(* Logix 5000 project; controller CLASE_1 Emulate 5570 rev 28.11; software revision 28.02; part 13 of 15 *)
(* tags used below, declared in another part *)
   Ref_FaultCodeList : P_DescList[1];   // Tag containing List of Fault Codes (DINT) and their Descriptions (STRING)
   Inp_LastFaultCode : DINT;   // Most recent drive fault code (enumeration)
   Inp_Ready : BOOL;   // 1=Drive is ready to run
   Inp_CommandDir : BOOL;   // 1=Drive is commanded Forward, 0=Drive is commanded Reverse
   Inp_ActualDir : BOOL;   // 1=Drive is running Forward, 0=Drive is running Reverse
   Inp_FwdPermOK : BOOL;   // 1=Permissives OK, drive can start Forward
   Inp_FwdNBPermOK : BOOL;   // 1=Non-Bypassable Permissives OK, drive can start Forward
   Inp_RevPermOK : BOOL;   // 1=Permissives OK, drive can start Reverse
   Inp_RevNBPermOK : BOOL;   // 1=Non-Bypassable Permissives OK, motor can start Reverse
   Inp_IntlkOK : BOOL;   // 1=Interlocks OK, drive can start/run
   Inp_NBIntlkOK : BOOL;   // 1=Non-Bypassable Interlocks OK, drive can start/run
   Inp_IOFault : BOOL;   // Input Communication Status 0=OK, 1=fail
   Inp_Sim : BOOL;   // 1=Simulate working drive; 0=Start/Stop/ Monitor actual drive
   Inp_OvrdCmd : SINT;   // Override Mode Command: 0=None, 1=Stop, 2=Start Fwd 3=Start Rev
   Cfg_HasJog : BOOL;   // 1=Drive Jog Command enabled/visible, 0=Drive Jog Command not allowed
   Cfg_HasRunFdbk : BOOL;   // 1=Drive provides feedback signal on Inp_Running when running
   Cfg_UseRunFdbk : BOOL;   // 1=Drive run feedback should be used for failure checking
   Cfg_HasSpeedFdbk : BOOL;   // 1=Drive provides speed feedback on Inp_SpeedFdbk
   Cfg_UseSpeedFdbk : BOOL;   // 1=Drive speed determines running state, 0=state determined by drive Active input bit
   Cfg_HasOutDatalink : BOOL;   // 1=A signal is connected to Out_Datalink
   Cfg_SetTrack : BOOL;   // 1=PSets track OSets in Oper, OSets track PSets in Prog, 0=no tracking
   Cfg_SetTrackOvrdHand : BOOL;   // 1=Prog/Oper Settings track Override/Hand speed reference
   Cfg_PCmdClear : ALIAS FOR Mode.Cfg_PCmdClear;
   Cfg_ProgDefault : ALIAS FOR Mode.Cfg_ProgDefault;
   Cfg_OperStopPrio : BOOL;   // 1=OCmd_Stop has priority, accepted any time, 0=OCmd_Stop only in Oper, Maint Mode.
   Cfg_OCmdResets : BOOL;   // 1=New Oper drive cmd. resets fault, 0=reset req'd to clear fault
   Cfg_ShedOnFailToStart : BOOL;   // 1=Stop Motor and Alarm on Fail to Start; 0=Alarm only on Fail to Start
   Cfg_ShedOnIOFault : BOOL;   // 1=Stop Motor and Alarm on I/O Fault; 0=Alarm only on I/O Fault
   Cfg_FailToStartAckReqd : ALIAS FOR FailToStart.Cfg_AckReqd;   // 1=Acknowledge required for Fail to Start Alarm
   Cfg_FailToStopAckReqd : ALIAS FOR FailToStop.Cfg_AckReqd;   // 1=Acknowledge required for Fail to Stop Alarm
   Cfg_IntlkTripAckReqd : ALIAS FOR IntlkTrip.Cfg_AckReqd;   // 1=Acknowledge required for Interlock Trip Alarm
   Cfg_DriveFaultAckReqd : ALIAS FOR DriveFault.Cfg_AckReqd;   // 1=Acknowledge required for Drive Fault Alarm
   Cfg_IOFaultAckReqd : ALIAS FOR IOFault.Cfg_AckReqd;   // 1=Acknowledge required for I/O Fault Alarm
   Cfg_FailToStartSeverity : ALIAS FOR FailToStart.Cfg_Severity;   // Fail To Start Alarm Severity: 1..250=Low, 251..500=Medium, 501..750=High, 751..1000=Urgent
   Cfg_FailToStopSeverity : ALIAS FOR FailToStop.Cfg_Severity;   // Fail To Stop Alarm Severity: 1..250=Low, 251..500=Medium, 501..750=High, 751..1000=Urgent
   Cfg_IntlkTripSeverity : ALIAS FOR IntlkTrip.Cfg_Severity;   // Interlock Trip Alarm Severity: 1..250=Low, 251..500=Medium, 501..750=High, 751..1000=Urgent
   Cfg_DriveFaultSeverity : ALIAS FOR DriveFault.Cfg_Severity;   // Drive Fault Alarm Severity: 1..250=Low, 251..500=Medium, 501..750=High, 751..1000=Urgent
   Cfg_IOFaultSeverity : ALIAS FOR IOFault.Cfg_Severity;   // I/O Fault Alarm Severity: 1..250=Low, 251..500=Medium, 501..750=High, 751..1000=Urgent
   Cfg_MinSpdRef : REAL;   // Minimum Speed Reference in EU (for limiting)
   Cfg_MaxSpdRef : REAL;   // Maximum Speed Reference in EU (for limiting)
   Cfg_SpeedRefRawMin : REAL;   // Speed Reference Minimum in Drive (raw) Units (for scaling)
   Cfg_SpeedRefRawMax : REAL;   // Speed Reference Maximum in Drive (raw) Units (for scaling)
   Cfg_SpeedRefEUMin : REAL;   // Speed Reference Minimum in Engineering Units (for scaling)
   Cfg_SpeedRefEUMax : REAL;   // Speed Reference Maximum in Engineering Units (for scaling)
   Cfg_SpeedFdbkRawMax : REAL;   // Speed Feedback Maximum in Drive (raw) Units (for scaling)
   Cfg_SpeedFdbkEUMax : REAL;   // Speed Feedback Maximum in Engineering Units (for scaling)
   Cfg_InpDatalinkRawMax : REAL;   // Input Datalink Maximum in Drive (raw) Units (for scaling)
   Cfg_InpDatalinkEUMax : REAL;   // Input Datalink Maximum in Engineering Units (for scaling)
   Cfg_OutDatalinkMax : REAL;   // Maximum Output Datalink in EU (for limiting)
   Cfg_OutDatalinkRawMin : REAL;   // Output Datalink Minimum in Drive (raw) Units (for scaling)
   Cfg_OutDatalinkRawMax : REAL;   // Output Datalink Maximum in Drive (raw) Units (for scaling)
   Cfg_OutDatalinkEUMin : REAL;   // Output Datalink Minimum in Engineering Units (for scaling)
   Cfg_OutDatalinkEUMax : REAL;   // Output Datalink Maximum in Engineering Units (for scaling)
   Cfg_SimRampT : DINT;   // Time to ramp speed fdbk when in Simulation (sec)
   Cfg_FailToStartT : DINT;   // Time after Start to get Run Feedback before Fault (sec)
   Cfg_FailToStopT : DINT;   // Time after Stop to drop Run Feedback before Fault (sec)
   Cfg_ResetPulseT : DINT;   // Time to pulse Out_Reset to clear drive fault
   Cfg_OperKeep : SINT;   // Oper keeps control in Prog Mode: .0=Reference, .1=Start/Stop, .2=Fwd/Rev, .3=OutDatalink
   Cfg_ProgKeep : SINT;   // Prog keeps control in Oper Mode: .0=Reference, .1=Start/Stop, .2=Fwd/Rev, .3=OutDatalink
   PSet_SpeedRef : REAL;   // Program Setting of Speed Reference (EU)
   PSet_OutDatalink : REAL;   // Program Setting of Output Datalink (EU)
   PSet_Owner : DINT;   // Program Owner Request ID (non-zero) or Release (zero)
   OSet_SpeedRef : REAL;   // Operator Setting of Speed Reference (EU)
   OSet_OutDatalink : REAL;   // Operator Setting of Output Datalink (EU)
   PCmd_Start : BOOL;   // Program Command to Start Drive
   PCmd_Stop : BOOL;   // Program Command to Stop Drive
   PCmd_Fwd : BOOL;   // Program Command to set direction to Fowrard
   PCmd_Rev : BOOL;   // Program Command to set direction to Reverse
   PCmd_Reset : BOOL;   // Program Command to Reset drive fault and all Alarms requiring Reset
   OCmd_Start : BOOL;   // Operator Command to Start Drive
   OCmd_Stop : BOOL;   // Operator Command to Stop Drive
   OCmd_Jog : BOOL;   // Operator Command to Jog Drive (not cleared by P_VSD!)
   OCmd_Fwd : BOOL;   // Operator Command to set direction to Forward
   OCmd_Rev : BOOL;   // Operator Command to set direction to Reverse
   OCmd_Bypass : BOOL;   // Operator Command to Bypass all Bypassable Interlocks and Permissives
   OCmd_Check : BOOL;   // Operator Command to Check (not bypass) all Interlocks and Permissives
   MCmd_Disable : BOOL;   // Maintenance Command to Disable Drive
   MCmd_Enable : BOOL;   // Maintenance Command to Enable (allow to run) Drive
   OCmd_Reset : BOOL;   // Operator Command to Reset all Alarms requiring Reset
   OCmd_ResetAckAll : BOOL;   // Operator Command to Reset all Alarms and latched Shed conditions
   Out_SpeedRef : REAL;   // Drive Speed Reference in Drive Units (typ. 0-32767 = 0 to max freq.)
   Out_Datalink : REAL;   // Auxiliary Signal (datalink) Output in Drive (raw) Units
   Out_Run : BOOL;   // 1=Start/Run Drive, 0=Stop Drive (for held starter type)
   Out_Stop : BOOL;   // 1=Stop Drive, 0=drive left in current state
   Out_Start : BOOL;   // 1=Start Drive, 0=drive left in current state
   Out_Jog : BOOL;   // 1=Jog drive at Jog Speed, -->0=stop jogging
   Out_ClearFault : BOOL;   // 1=Attempt to clear Drive Fault
   Out_Fwd : BOOL;   // 1=Set drive direction to Forward
   Out_Rev : BOOL;   // 1=Set drive direction to Reverse
   Val_SpeedRef : REAL;   // Speed Reference (target) to drive
   Val_OutDatalink : REAL;   // Output Datalink value to drive
   Val_SpeedRefEUMax : REAL;   // Maximum of Speed Reference = MAX (Cfg_SpeedFdbkEUMin, Cfg_SpeedFdbkEUMax)
   Val_SpeedFdbkEUMax : REAL;   // Maximum of Speed Feedback = MAX (Cfg_SpeedFdbkEUMin, Cfg_SpeedFdbkEUMax)
   Val_LastFaultCode : DINT;   // Most recent drive fault code (enumeration)
   SrcQ_IO : SINT;   // Source and Quality of primary I/O (enumeration)
   SrcQ : SINT;   // Source and Quality of primary Val/Sts (enumeration)
   Val_Cmd : SINT;   // Device Command 0=None, 1=Stop, 2=StartFwd 3=StartRev 4=JogFwd 5=JogRev
   Val_Fdbk : SINT;   // Device Feedback 0=Stopped, 1=Running Fwd 2=Running Rev 3=Accelerating 4=Decelerating
   Val_Sts : SINT;   // Device Confirmed Sts 0? 1=Stop 2=RunF 3=RunR 4=JogF 5=JogR 6=Stopping 7=Starting F 8=Starting R, 33=Disabled
   Val_Fault : SINT;   // Device Fault Status 0=None, 16=Fail to Start, 17 = Fail to Stop, 18=Drive Fault, 32=I/O Fault, 34=Config Error
   Val_Mode : ALIAS FOR Mode.Val;
   Val_Owner : DINT;   // Current Object Owner ID (0=not owned)
   Val_Notify : SINT;   // Current Alarm Level and Acknowledgement (enumeration)
   Sts_Stopped : BOOL;   // 1=Drive requested to stop and is confirmed stopped
   Sts_Starting : BOOL;   // 1=Drive requested to run and awaiting run feedback
   Sts_Running : BOOL;   // 1=Drive requested to run and is confirmed running
   Sts_Stopping : BOOL;   // 1=Drive requested to stop and awaiting stopped feedback
   Sts_Jogging : BOOL;   // 1=Drive requested to Jog
   Sts_CommandDir : BOOL;   // 1=Drive commanded to Forward, 0=Reverse
   Sts_ActualDir : BOOL;   // 1=Drive Actual direction is Forward, 0=Reverse
   Sts_SpeedLimited : BOOL;   // 1=Speed Reference Setting exceeds configured Max/Min limit
   Sts_Disabled : BOOL;   // 1=Drive is Disabled
   Sts_NotRdy : BOOL;   // 1=Device Not Ready, see detail bits for reason
   Nrdy_OperPrio : BOOL;   // 1=Device Not Ready: Operator State 0 Priority Command Requires Reset
   Nrdy_Fail : BOOL;   // 1=Device Not Ready: Device Failure (Shed Requires Reset)
   Nrdy_IOFault : BOOL;   // 1=Device Not Ready: I/O Fault (Shed Requires Reset)
   Nrdy_Trip : BOOL;   // 1=Device not Ready: Deivce Tripped (Drive Fault)
   Sts_AlmInh : BOOL;   // 1=An Alarm is Shelved, Disabled or Suppressed, display icon
   Sts_Err : BOOL;   // 1=Error in Config: see detail bits for reason
   Err_FdbkRaw : BOOL;   // 1=Erron in Config: Speed Fdbk Raw Min = Max
   Err_FdbkEU : BOOL;   // 1=Error in Config: Speed Fdbk EU Min = Max
   Err_RefEU : BOOL;   // 1=Error in Config: Speed Ref EU Min = Max
   Err_OutDLEU : BOOL;   // 1=Error in Config: Output Datalink EU Min = Max
   Sts_Hand : ALIAS FOR Mode.Sts_Hand;
   Sts_Maint : ALIAS FOR Mode.Sts_Maint;
   Sts_Ovrd : ALIAS FOR Mode.Sts_Ovrd;
   Sts_Prog : ALIAS FOR Mode.Sts_Prog;
   Sts_Oper : ALIAS FOR Mode.Sts_Oper;
   Ack_FailToStart : ALIAS FOR FailToStart.Ack;   // 1=Fail to Start Alarm has been acknowledged
   Sts_FailToStop : ALIAS FOR FailToStop.Inp;   // 1=Drive Failed to Stop
   Ack_FailToStop : ALIAS FOR FailToStop.Ack;   // 1=Fail to Stop Alarm has been acknowledged
   Ack_IntlkTrip : ALIAS FOR IntlkTrip.Ack;   // 1=Interlock Trip Alarm has been acknowledged
   Sts_DriveFault : ALIAS FOR DriveFault.Inp;   // 1=Drive Fault (see drive display or manual)
   Ack_DriveFault : ALIAS FOR DriveFault.Ack;   // 1=Drive Fault Alarm has been acknowledged
   Sts_IOFault : ALIAS FOR IOFault.Inp;   // I/O Comm Fault Status (0=OK, 1=Bad)
   Ack_IOFault : ALIAS FOR IOFault.Ack;   // 1=I/O Fault Alarm has been acknowledged
   Rdy_Start : BOOL;   // 1=Ready to receive OCmd_Start (enables HMI button)
   Rdy_Stop : BOOL;   // 1=Ready to receive OCmd_Stop (enables HMI button)
   Rdy_Jog : BOOL;   // 1=Ready to receive OCmd_Jog (enables HMI button)
   Rdy_Bypass : BOOL;   // 1=Ready to receive OCmd_Bypass (enables HMI button)
   Rdy_Reset : BOOL;   // 1=Ready to receive OCmd_Reset (enables HMI button)
   Rdy_ResetAckAll : BOOL;   // 1=At least one Alarm or latched Shed condition requires Reset or Ack
   Rdy_SpeedRef : BOOL;   // 1=Ready to receive OSet_SpeedRef (enables data entry field)
   Rdy_OSet : BOOL;   // 1=Ready to receive OSets (other than CV) (enables data entry fields)
   P_VSD : BOOL;   // Unique Parameter Name for auto - discovery
   Mode : P_Mode;   // Drive Mode Selection
   IOFault : P_Alarm;   // I/O Fault Alarm
   IntlkTrip : P_Alarm;   // Interlock Trip Alarm
   FailToStop : P_Alarm;   // Drive Failed to Stop Alarm
   FailToStart : P_Alarm;   // Drive Failed to Start Alarm
   Wrk_Run : BOOL;   // 1=Drive should be "running", 0=should be "stopped"
   Wrk_RunFdbk : BOOL;   // Run Feedback based on mode, simulation, etc. 1=running
   Wrk_Notify : DINT;   // Buffer for building Val_Notify
   DriveFault : P_Alarm;   // Drive Faulted Alarm
   Wrk_SpeedRef : REAL;   // Working copy of Speed Reference (for limiting)
   Wrk_Rev : BOOL;   // Working (internal) Direction 1=Reverse 0=Forward (default)
   Wrk_Jog : BOOL;   // 1=Jog Drive, 0=Drive not jogging
   Wrk_OutDatalink : REAL;   // Selected Output Datalink setting
   Wrk_Cmd : SINT;   // Buffer for building Val_Cmd
   Wrk_Sts : SINT;   // Buffer for building Val_Sts
   Wrk_Fault : SINT;   // Buffer for building Val_Fault
   Wrk_Retrigger : BOOL;   // Maint Start issued while running or Stop while stopped
   Wrk_FaultDescFSC : CONTROL;   // FSC control for Fault Code List search
   Val_FaultDesc : STRING_40;   // Description of Drive Fault (given LastFaultCode)
   Wrk_SrcQ : SINT;   // Register for building Source / Quality enumeration
   Wrk_NotRdy : BOOL;   // Device Not Ready conditions excluding shed latches
(* P_VSD, continued *)

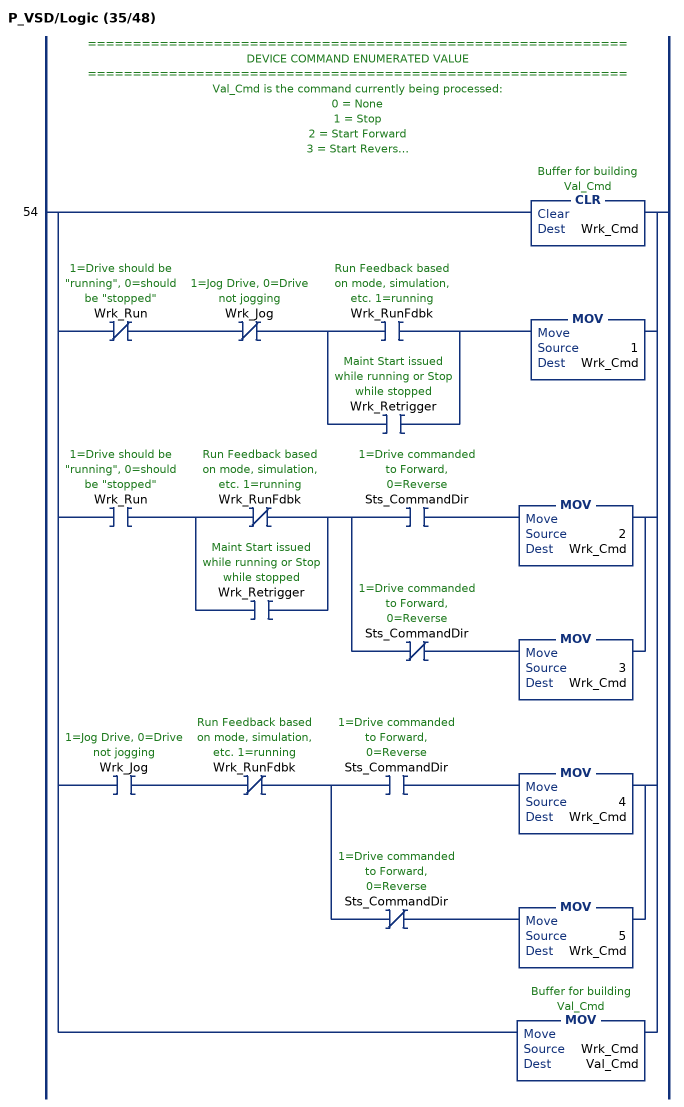
   [picture p271: P_VSD/Logic rungs 54-54]
   // ============================================================
   // DEVICE COMMAND ENUMERATED VALUE
   // ============================================================
   // Val_Cmd is the command currently being processed:
   // 0 = None
   // 1 = Stop
   // 2 = Start Forward
   // 3 = Start Reverse
   // 4 = Jog Forward
   // 5 = Jog Reverse
   54: [CLR(Wrk_Cmd) ,XIO(Wrk_Run) XIO(Wrk_Jog) [XIC(Wrk_RunFdbk) ,XIC(Wrk_Retrigger) ] MOV(1,Wrk_Cmd) ,XIC(Wrk_Run) [XIO(Wrk_RunFdbk) ,XIC(Wrk_Retrigger) ] [XIC(Sts_CommandDir) MOV(2,Wrk_Cmd) ,XIO(Sts_CommandDir) MOV(3,Wrk_Cmd) ] ,XIC(Wrk_Jog) XIO(Wrk_RunFdbk) [XIC(Sts_CommandDir) MOV(4,Wrk_Cmd) ,XIO(Sts_CommandDir) MOV(5,Wrk_Cmd) ] ,MOV(Wrk_Cmd,Val_Cmd) ];
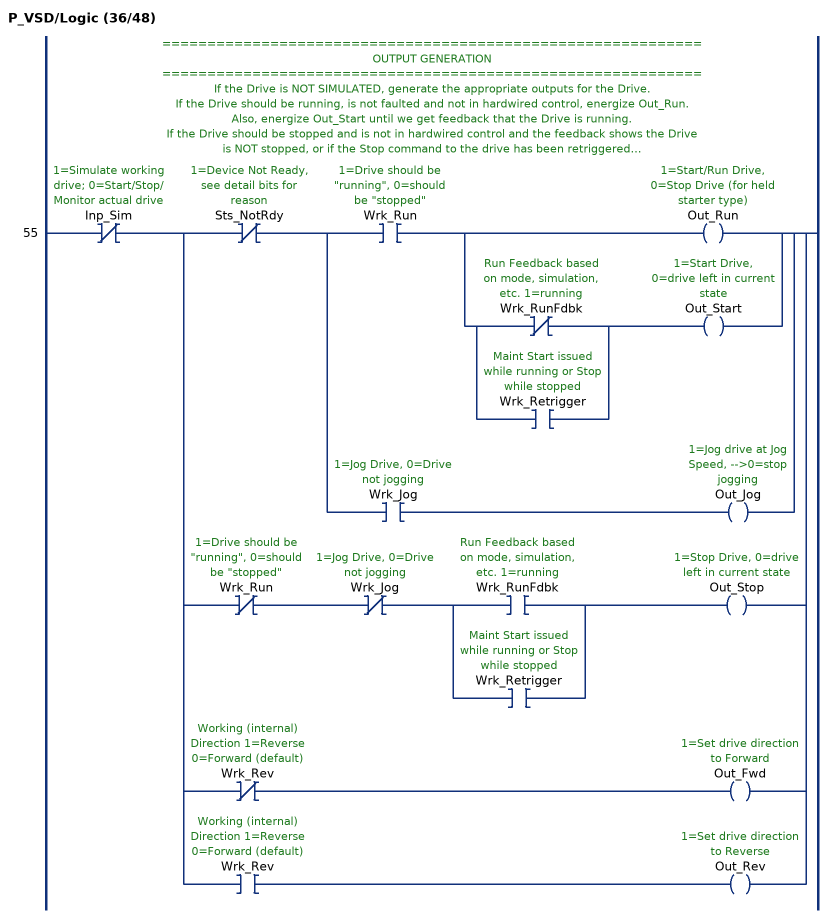
   // ============================================================
   // OUTPUT GENERATION
   // ============================================================
   // If the Drive is NOT SIMULATED, generate the appropriate outputs for the Drive.
   // If the Drive should be running, is not faulted and not in hardwired control, energize Out_Run.
   // Also, energize Out_Start until we get feedback that the Drive is running.
   // If the Drive should be stopped and is not in hardwired control and the feedback shows the Drive
   // is NOT stopped, or if the Stop command to the drive has been retriggered,
   // energize the Out_Stop output to stop the Drive.
   // Finally, if the drive is not simulated, energize the appropriate direction output.
   // #####  V3.5-02  2016-03-22:  Modified to eliminate oscillating Out_Stop on Drive Not Ready.  #####
   55: XIO(Inp_Sim)[XIO(Sts_NotRdy) [XIC(Wrk_Run) [OTE(Out_Run) ,[XIO(Wrk_RunFdbk) ,XIC(Wrk_Retrigger) ] OTE(Out_Start) ] ,XIC(Wrk_Jog) OTE(Out_Jog) ] ,XIO(Wrk_Run) XIO(Wrk_Jog) [XIC(Wrk_RunFdbk) ,XIC(Wrk_Retrigger) ] OTE(Out_Stop) ,XIO(Wrk_Rev) OTE(Out_Fwd) ,XIC(Wrk_Rev) OTE(Out_Rev) ];
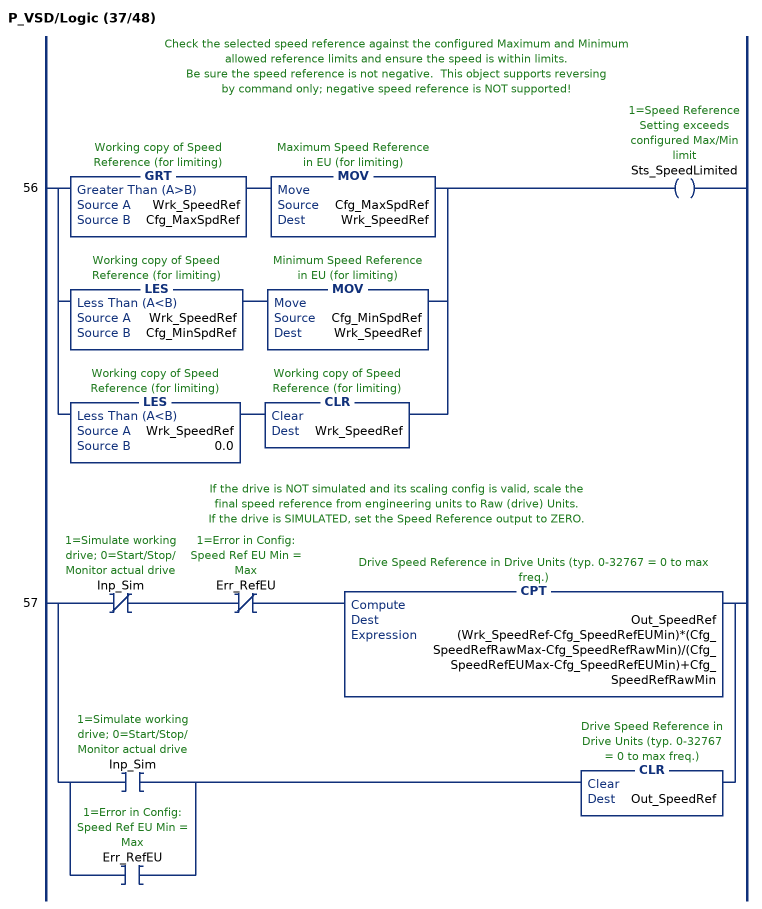
   // Check the selected speed reference against the configured Maximum and Minimum
   // allowed reference limits and ensure the speed is within limits.
   // Be sure the speed reference is not negative.  This object supports reversing
   // by command only; negative speed reference is NOT supported!
   56: [GRT(Wrk_SpeedRef,Cfg_MaxSpdRef) MOV(Cfg_MaxSpdRef,Wrk_SpeedRef) ,LES(Wrk_SpeedRef,Cfg_MinSpdRef) MOV(Cfg_MinSpdRef,Wrk_SpeedRef) ,LES(Wrk_SpeedRef,0.0) CLR(Wrk_SpeedRef) ]OTE(Sts_SpeedLimited);
   // If the drive is NOT simulated and its scaling config is valid, scale the
   // final speed reference from engineering units to Raw (drive) Units.
   // If the drive is SIMULATED, set the Speed Reference output to ZERO.
   57: [XIO(Inp_Sim) XIO(Err_RefEU) CPT(Out_SpeedRef,(Wrk_SpeedRef-Cfg_SpeedRefEUMin)*(Cfg_SpeedRefRawMax-Cfg_SpeedRefRawMin)/(Cfg_SpeedRefEUMax-Cfg_SpeedRefEUMin)+Cfg_SpeedRefRawMin) ,[XIC(Inp_Sim) ,XIC(Err_RefEU) ] CLR(Out_SpeedRef) ];
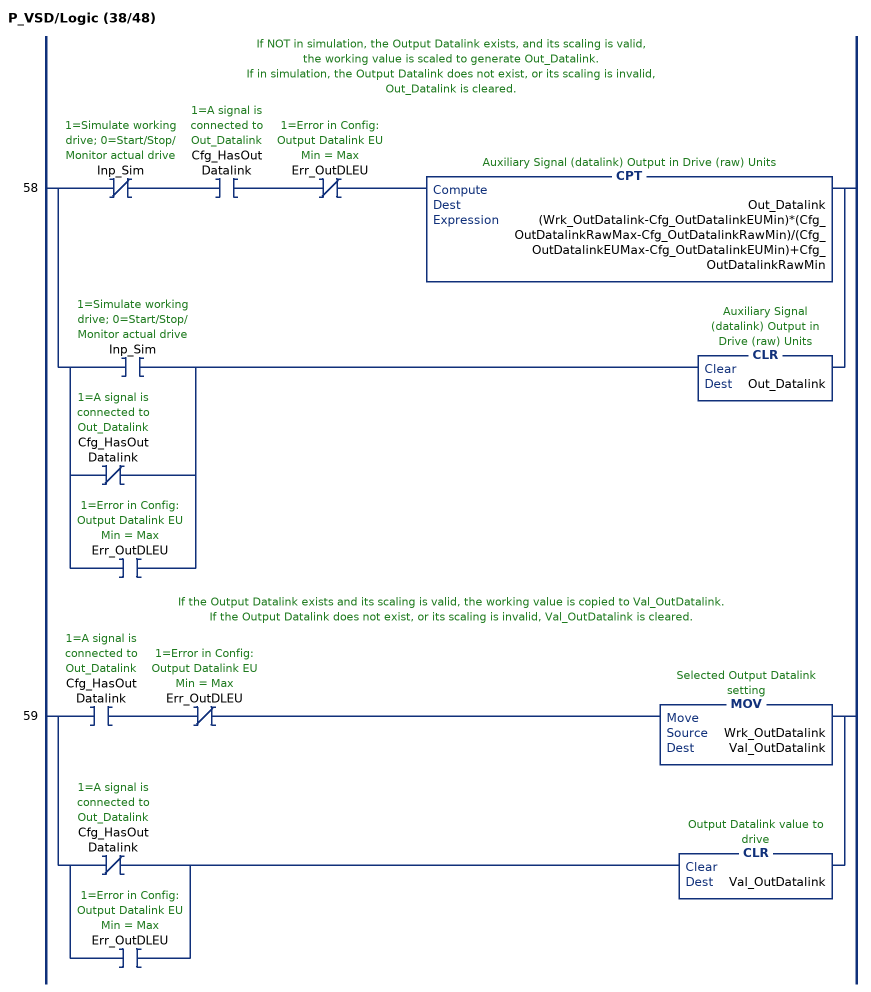
   // If NOT in simulation, the Output Datalink exists, and its scaling is valid,
   // the working value is scaled to generate Out_Datalink.
   // If in simulation, the Output Datalink does not exist, or its scaling is invalid,
   // Out_Datalink is cleared.
   58: [XIO(Inp_Sim) XIC(Cfg_HasOutDatalink) XIO(Err_OutDLEU) CPT(Out_Datalink,(Wrk_OutDatalink-Cfg_OutDatalinkEUMin)*(Cfg_OutDatalinkRawMax-Cfg_OutDatalinkRawMin)/(Cfg_OutDatalinkEUMax-Cfg_OutDatalinkEUMin)+Cfg_OutDatalinkRawMin) ,[XIC(Inp_Sim) ,XIO(Cfg_HasOutDatalink) ,XIC(Err_OutDLEU) ] CLR(Out_Datalink) ];
   // If the Output Datalink exists and its scaling is valid, the working value is copied to Val_OutDatalink.
   // If the Output Datalink does not exist, or its scaling is invalid, Val_OutDatalink is cleared.
   59: [XIC(Cfg_HasOutDatalink) XIO(Err_OutDLEU) MOV(Wrk_OutDatalink,Val_OutDatalink) ,[XIO(Cfg_HasOutDatalink) ,XIC(Err_OutDLEU) ] CLR(Val_OutDatalink) ];
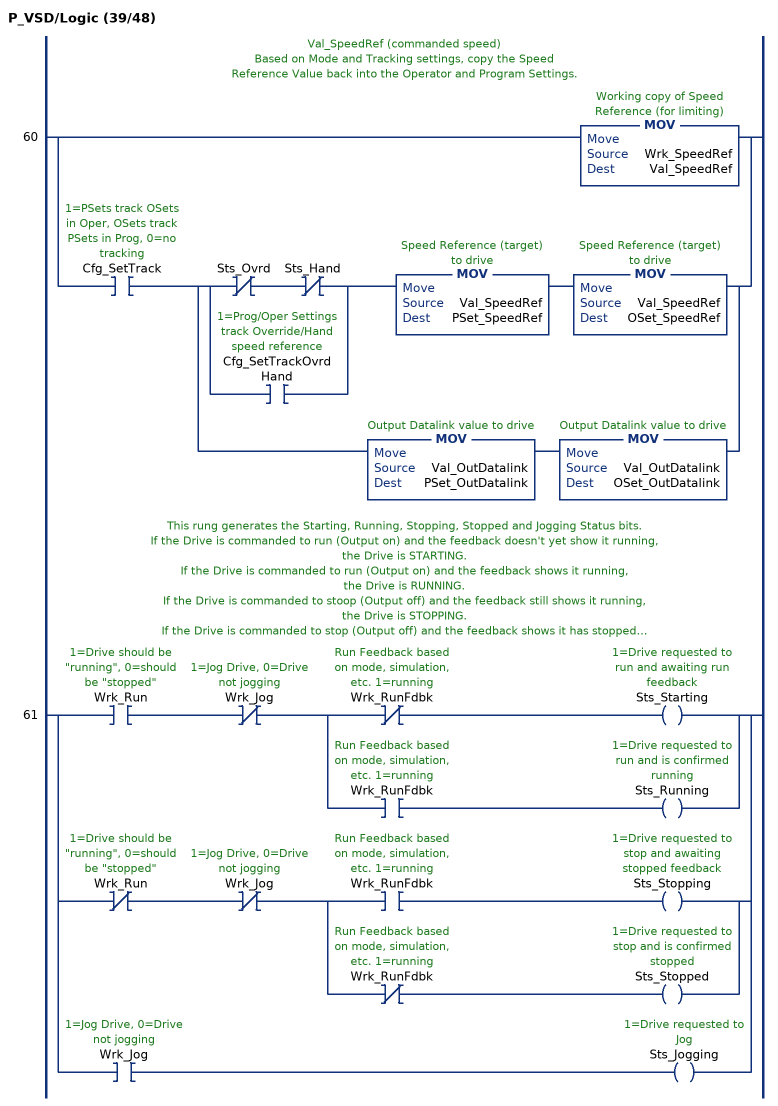
   // Val_SpeedRef (commanded speed)
   // Based on Mode and Tracking settings, copy the Speed
   // Reference Value back into the Operator and Program Settings.
   60: [MOV(Wrk_SpeedRef,Val_SpeedRef) ,XIC(Cfg_SetTrack) [[XIO(Sts_Ovrd) XIO(Sts_Hand) ,XIC(Cfg_SetTrackOvrdHand) ] MOV(Val_SpeedRef,PSet_SpeedRef) MOV(Val_SpeedRef,OSet_SpeedRef) ,MOV(Val_OutDatalink,PSet_OutDatalink) MOV(Val_OutDatalink,OSet_OutDatalink) ] ];
   // This rung generates the Starting, Running, Stopping, Stopped and Jogging Status bits.
   // If the Drive is commanded to run (Output on) and the feedback doesn't yet show it running,
   // the Drive is STARTING.
   // If the Drive is commanded to run (Output on) and the feedback shows it running,
   // the Drive is RUNNING.
   // If the Drive is commanded to stoop (Output off) and the feedback still shows it running,
   // the Drive is STOPPING.
   // If the Drive is commanded to stop (Output off) and the feedback shows it has stopped,
   // the Drive is STOPPED.
   // #####  V3.0-00  2013-06-30:  Removed check of Cfg_UseRunFdbk --  #####
   // #####  now uses run feedback  based on speed fdbk  #####
   61: [XIC(Wrk_Run) XIO(Wrk_Jog) [XIO(Wrk_RunFdbk) OTE(Sts_Starting) ,XIC(Wrk_RunFdbk) OTE(Sts_Running) ] ,XIO(Wrk_Run) XIO(Wrk_Jog) [XIC(Wrk_RunFdbk) OTE(Sts_Stopping) ,XIO(Wrk_RunFdbk) OTE(Sts_Stopped) ] ,XIC(Wrk_Jog) OTE(Sts_Jogging) ];
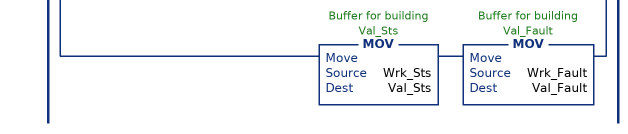
   // Val_Sts is the current device status, as determined by this AOI,
   // based on its knowledge of commands executed and feedback.
   // (This is the status that should be monitored by, for example, FT Historian.)
   // 0 = Powerup / Unknown (Hand Mode with no feedback, for example)
   // 1 = Stopped
   // 2 = Running Forward
   // 3 = Running Reverse
   // 4 = Jogging Forward
   // 5 = Jogging Reverse
   // 6 = Stopping
   // 7 = Starting Forward
   // 8 = Starting Reverse
   // 33 = Device Disabled
   // Val_Fault is the current device fault status, as determined by this AOI,
   // based on its knowledge of commands executed and feedback.
   // (This is the fault status that should be monitored by, for example, FT Historian.)
   // 0 = None
   // 16 = Fail to Start
   // 17 = Fail to Stop
   // 18 = Drive Fault
   // 32 = I/O Fault (from Input)
   // 34 = Configuration Error
   // #####  V3.1-00  2014-06-30: Added Not Ready reason bits (Nrdy_xxx)  #####
   62: [CLR(Wrk_Sts) CLR(Wrk_Fault) ,XIC(Sts_Stopped) MOV(1,Wrk_Sts) ,XIC(Sts_Running) [XIC(Sts_ActualDir) MOV(2,Wrk_Sts) ,XIO(Sts_ActualDir) MOV(3,Wrk_Sts) ] ,XIC(Sts_Jogging) [XIC(Sts_ActualDir) MOV(4,Wrk_Sts) ,XIO(Sts_ActualDir) MOV(5,Wrk_Sts) ] ,XIC(Sts_Stopping) MOV(6,Wrk_Sts) ,XIC(Sts_Starting) [XIC(Sts_CommandDir) MOV(7,Wrk_Sts) ,XIO(Sts_CommandDir) MOV(8,Wrk_Sts) ] ,XIC(Nrdy_Fail) MOV(16,Wrk_Fault) ,XIC(Sts_FailToStop) MOV(17,Wrk_Fault) ,XIC(Sts_DriveFault) MOV(18,Wrk_Fault) ,XIC(Nrdy_IOFault) MOV(32,Wrk_Fault) ,XIC(Sts_Disabled) MOV(33,Wrk_Sts) ,XIC(Sts_Err) MOV(34,Wrk_Fault) ,MOV(Wrk_Sts,Val_Sts) MOV(Wrk_Fault,Val_Fault) ];
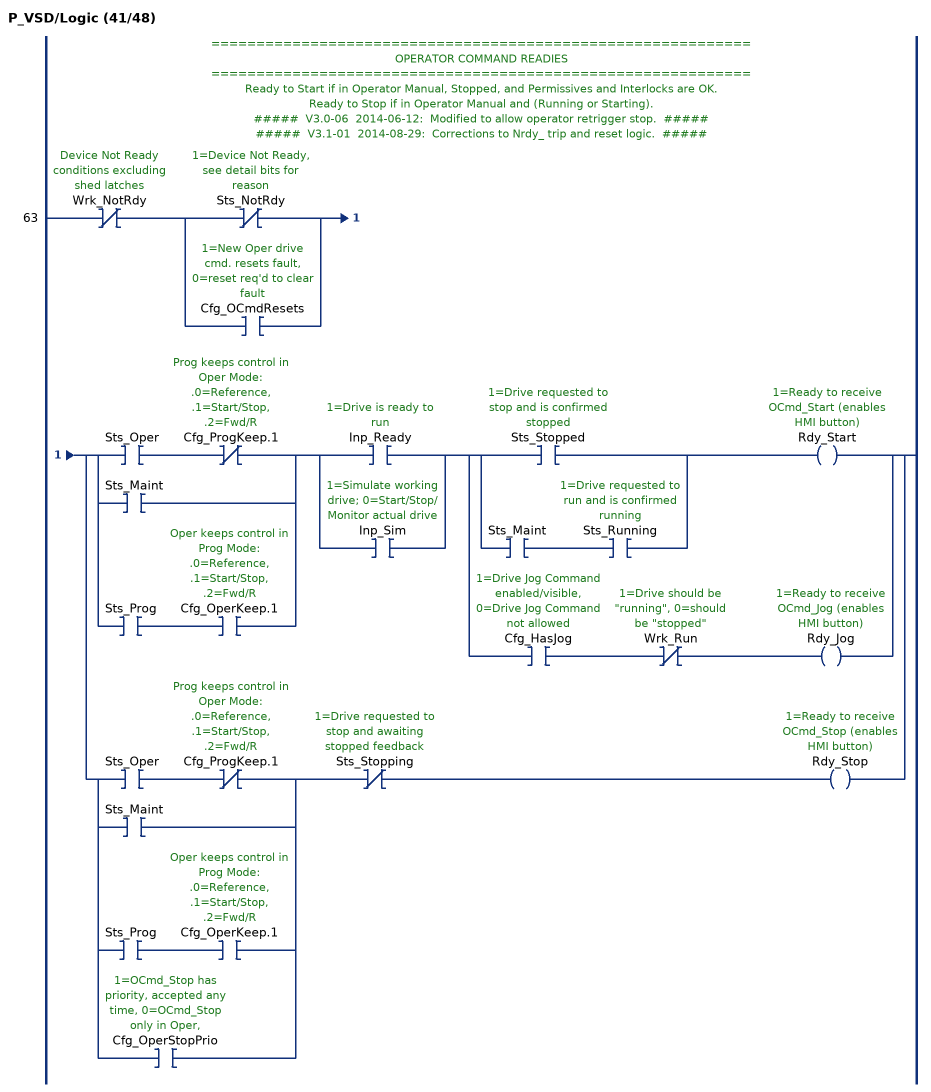
   // ============================================================
   // OPERATOR COMMAND READIES
   // ============================================================
   // Ready to Start if in Operator Manual, Stopped, and Permissives and Interlocks are OK.
   // Ready to Stop if in Operator Manual and (Running or Starting).
   // #####  V3.0-06  2014-06-12:  Modified to allow operator retrigger stop.  #####
   // #####  V3.1-01  2014-08-29:  Corrections to Nrdy_ trip and reset logic.  #####
   63: XIO(Wrk_NotRdy)[XIO(Sts_NotRdy) ,XIC(Cfg_OCmdResets) ][[XIC(Sts_Oper) XIO(Cfg_ProgKeep.1) ,XIC(Sts_Maint) ,XIC(Sts_Prog) XIC(Cfg_OperKeep.1) ] [XIC(Inp_Ready) ,XIC(Inp_Sim) ] [[XIC(Sts_Stopped) ,XIC(Sts_Maint) XIC(Sts_Running) ] OTE(Rdy_Start) ,XIC(Cfg_HasJog) XIO(Wrk_Run) OTE(Rdy_Jog) ] ,[XIC(Sts_Oper) XIO(Cfg_ProgKeep.1) ,XIC(Sts_Maint) ,XIC(Sts_Prog) XIC(Cfg_OperKeep.1) ,XIC(Cfg_OperStopPrio) ] XIO(Sts_Stopping) OTE(Rdy_Stop) ];
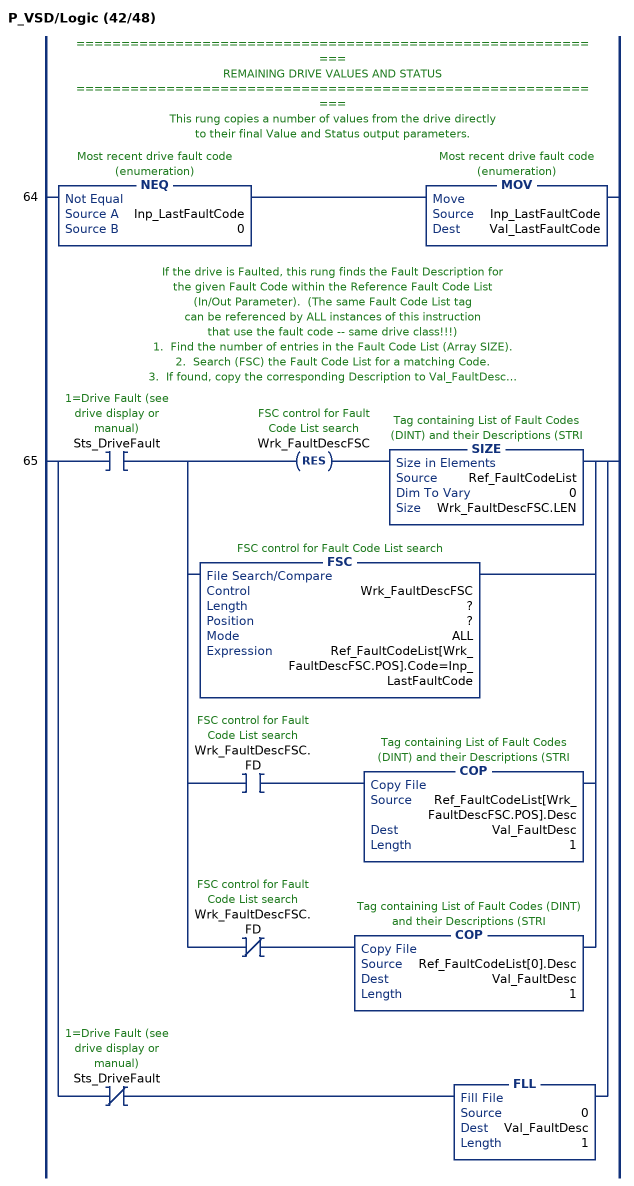
   // ============================================================
   // REMAINING DRIVE VALUES AND STATUS
   // ============================================================
   // This rung copies a number of values from the drive directly
   // to their final Value and Status output parameters.
   64: NEQ(Inp_LastFaultCode,0)MOV(Inp_LastFaultCode,Val_LastFaultCode);
   // If the drive is Faulted, this rung finds the Fault Description for
   // the given Fault Code within the Reference Fault Code List
   // (In/Out Parameter).  (The same Fault Code List tag
   // can be referenced by ALL instances of this instruction
   // that use the fault code -- same drive class!!!)
   // 1.  Find the number of entries in the Fault Code List (Array SIZE).
   // 2.  Search (FSC) the Fault Code List for a matching Code.
   // 3.  If found, copy the corresponding Description to Val_FaultDesc.
   // 4.  If NOT found, copy list entry zero ("No Help Available for this code").
   // And if the drive is not faulted, clear the Val_FaultDesc string.
   // #####  V3.0-00  2013-06-30:  Added rung  #####
   65: [XIC(Sts_DriveFault) [RES(Wrk_FaultDescFSC) SIZE(Ref_FaultCodeList,0,Wrk_FaultDescFSC.LEN) ,FSC(Wrk_FaultDescFSC,?,?,ALL,Ref_FaultCodeList[Wrk_FaultDescFSC.POS].Code=Inp_LastFaultCode) ,XIC(Wrk_FaultDescFSC.FD) COP(Ref_FaultCodeList[Wrk_FaultDescFSC.POS].Desc,Val_FaultDesc,1) ,XIO(Wrk_FaultDescFSC.FD) COP(Ref_FaultCodeList[0].Desc,Val_FaultDesc,1) ] ,XIO(Sts_DriveFault) FLL(0,Val_FaultDesc,1) ];
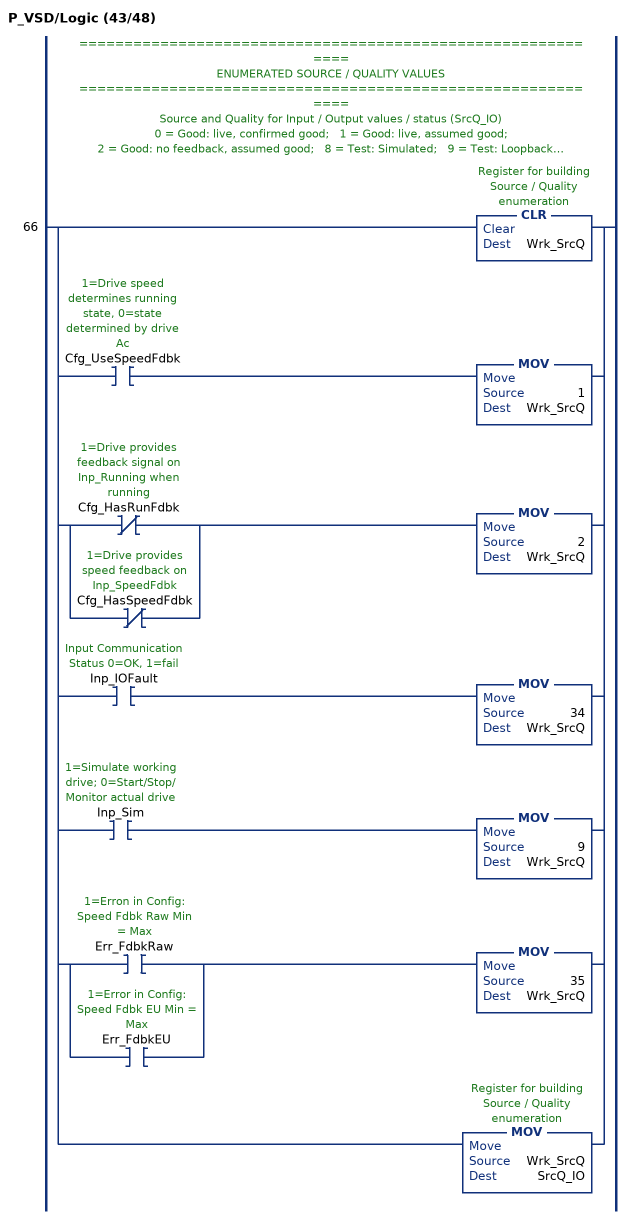
   // ============================================================
   // ENUMERATED SOURCE / QUALITY VALUES
   // ============================================================
   // Source and Quality for Input / Output values / status (SrcQ_IO)
   // 0 = Good: live, confirmed good;   1 = Good: live, assumed good;
   // 2 = Good: no feedback, assumed good;   8 = Test: Simulated;   9 = Test: Loopback;
   // 10 = Test: Manually Entered;   16 = Uncertain: Live, off-spec;
   // 17 = Uncertain, Substituted at Device / Bus;   18 = Uncertain, Substituted at AOI;
   // 19 = Uncertain, using last known good;    20 = Uncertain, using replacement value;
   // 32 = Bad, Signal Failure;   33 = Bad, Channel Fault;
   // 34 = Bad, Module / Comms Fault;   35 = Bad, Invalid Configuration
   // #####  V3.1-00  2014-06-30:  Added rung for Source/Quality enumerations.  #####
   // #####  V3.1-04 Patch01  2015-09-25:  Modified for correct meaning / handling of  #####
   // #####  Cfg_UseSpeedFdbk = 1 (state determined by speed), Cfg_HasRunFdbk = 0  #####
   // #####  (state assumed), and Cfg_HasSpeedFdbk = 0 (speed assumed, no feedback).  #####
   66: [CLR(Wrk_SrcQ) ,XIC(Cfg_UseSpeedFdbk) MOV(1,Wrk_SrcQ) ,[XIO(Cfg_HasRunFdbk) ,XIO(Cfg_HasSpeedFdbk) ] MOV(2,Wrk_SrcQ) ,XIC(Inp_IOFault) MOV(34,Wrk_SrcQ) ,XIC(Inp_Sim) MOV(9,Wrk_SrcQ) ,[XIC(Err_FdbkRaw) ,XIC(Err_FdbkEU) ] MOV(35,Wrk_SrcQ) ,MOV(Wrk_SrcQ,SrcQ_IO) ];
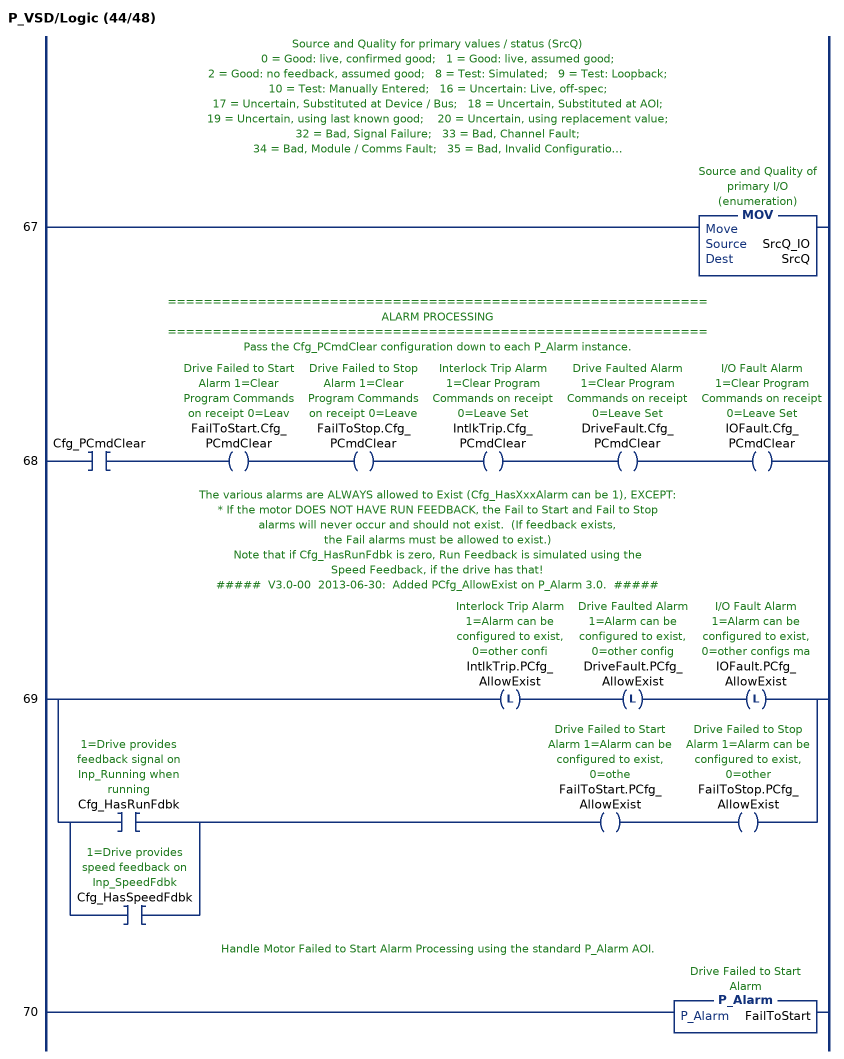
   // Source and Quality for primary values / status (SrcQ)
   // 0 = Good: live, confirmed good;   1 = Good: live, assumed good;
   // 2 = Good: no feedback, assumed good;   8 = Test: Simulated;   9 = Test: Loopback;
   // 10 = Test: Manually Entered;   16 = Uncertain: Live, off-spec;
   // 17 = Uncertain, Substituted at Device / Bus;   18 = Uncertain, Substituted at AOI;
   // 19 = Uncertain, using last known good;    20 = Uncertain, using replacement value;
   // 32 = Bad, Signal Failure;   33 = Bad, Channel Fault;
   // 34 = Bad, Module / Comms Fault;   35 = Bad, Invalid Configuration
   // If the drive is using run feedback (for state) and has speed feedback, all is live and good.
   // If the drive is using speed feedback to determine run state, state is assumed good.
   // If the drive does not have speed feedback, speed is no-feedback assumed good.
   // #####  V3.1-00  2014-06-30:  Added rung for Source/Quality enumerations.  #####
   // #####  V3.1-04 Patch01  2015-09-25:  Modified: instruction does not have substitution of speed feedback.  #####
   67: MOV(SrcQ_IO,SrcQ);
   // ============================================================
   // ALARM PROCESSING
   // ============================================================
   // Pass the Cfg_PCmdClear configuration down to each P_Alarm instance.
   68: XIC(Cfg_PCmdClear)OTE(FailToStart.Cfg_PCmdClear)OTE(FailToStop.Cfg_PCmdClear)OTE(IntlkTrip.Cfg_PCmdClear)OTE(DriveFault.Cfg_PCmdClear)OTE(IOFault.Cfg_PCmdClear);
   // The various alarms are ALWAYS allowed to Exist (Cfg_HasXxxAlarm can be 1), EXCEPT:
   // * If the motor DOES NOT HAVE RUN FEEDBACK, the Fail to Start and Fail to Stop
   // alarms will never occur and should not exist.  (If feedback exists,
   // the Fail alarms must be allowed to exist.)
   // Note that if Cfg_HasRunFdbk is zero, Run Feedback is simulated using the
   // Speed Feedback, if the drive has that!
   // #####  V3.0-00  2013-06-30:  Added PCfg_AllowExist on P_Alarm 3.0.  #####
   69: [OTL(IntlkTrip.PCfg_AllowExist) OTL(DriveFault.PCfg_AllowExist) OTL(IOFault.PCfg_AllowExist) ,[XIC(Cfg_HasRunFdbk) ,XIC(Cfg_HasSpeedFdbk) ] OTE(FailToStart.PCfg_AllowExist) OTE(FailToStop.PCfg_AllowExist) ];
   // Handle Motor Failed to Start Alarm Processing using the standard P_Alarm AOI.
   70: P_Alarm(FailToStart);
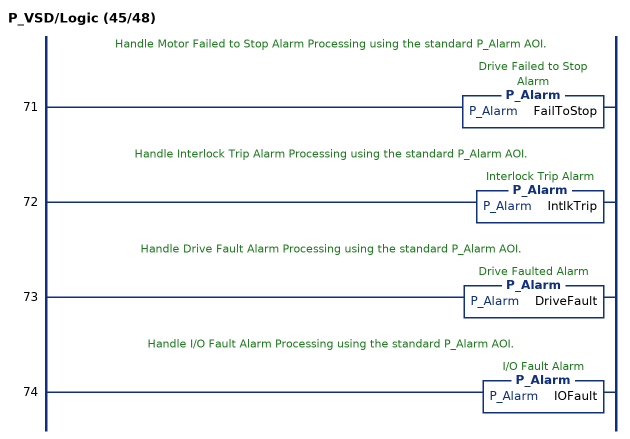
   // Handle Motor Failed to Stop Alarm Processing using the standard P_Alarm AOI.
   71: P_Alarm(FailToStop);
   // Handle Interlock Trip Alarm Processing using the standard P_Alarm AOI.
   72: P_Alarm(IntlkTrip);
   // Handle Drive Fault Alarm Processing using the standard P_Alarm AOI.
   73: P_Alarm(DriveFault);
   // Handle I/O Fault Alarm Processing using the standard P_Alarm AOI.
   74: P_Alarm(IOFault);
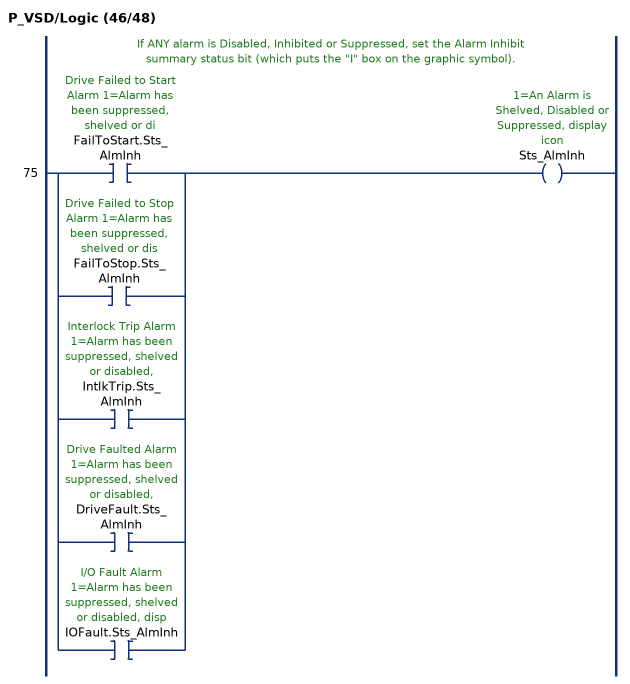
   // If ANY alarm is Disabled, Inhibited or Suppressed, set the Alarm Inhibit
   // summary status bit (which puts the "I" box on the graphic symbol).
   75: [XIC(FailToStart.Sts_AlmInh) ,XIC(FailToStop.Sts_AlmInh) ,XIC(IntlkTrip.Sts_AlmInh) ,XIC(DriveFault.Sts_AlmInh) ,XIC(IOFault.Sts_AlmInh) ]OTE(Sts_AlmInh);
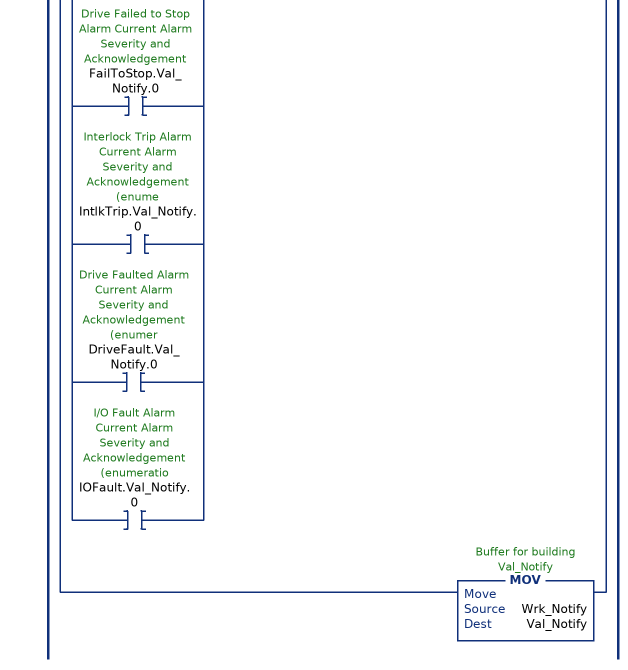
   // ============================================================
   // NOTIFICATION VALUE
   // ============================================================
   // Indicate the current alarm notification level as the max of any of the alarms,
   // and set the low-order bit for reset or ack required:
   // 0 = Not in alarm, acknowledged
   // 1 = Not in alarm, unacknowledged or reset required
   // 2 = Low severity alarm, acknowledged
   // 3 = Low severity alarm, unacknowledged
   // 4 = Medium severity alarm, acknowledged
   // 5 = Medium severity alarm, unacknowledged
   // 6 = High severity alarm, acknowledged
   // 7 = High severity alarm, unacknowledged
   // 8 = Urgent severity alarm, acknowledged
   // 9 = Urgent severity alarm, unacknowledged
   // #####  V3.1-00  2014-06-30:  Separated Reset Reqd functions from Val_Notify  #####
   76: [CLR(Wrk_Notify) ,GRT(FailToStart.Val_Notify,Wrk_Notify) MOV(FailToStart.Val_Notify,Wrk_Notify) ,GRT(FailToStop.Val_Notify,Wrk_Notify) MOV(FailToStop.Val_Notify,Wrk_Notify) ,GRT(IntlkTrip.Val_Notify,Wrk_Notify) MOV(IntlkTrip.Val_Notify,Wrk_Notify) ,GRT(DriveFault.Val_Notify,Wrk_Notify) MOV(DriveFault.Val_Notify,Wrk_Notify) ,GRT(IOFault.Val_Notify,Wrk_Notify) MOV(IOFault.Val_Notify,Wrk_Notify) ,[XIC(FailToStart.Val_Notify.0) ,XIC(FailToStop.Val_Notify.0) ,XIC(IntlkTrip.Val_Notify.0) ,XIC(DriveFault.Val_Notify.0) ,XIC(IOFault.Val_Notify.0) ] OTE(Wrk_Notify.0) ,MOV(Wrk_Notify,Val_Notify) ];
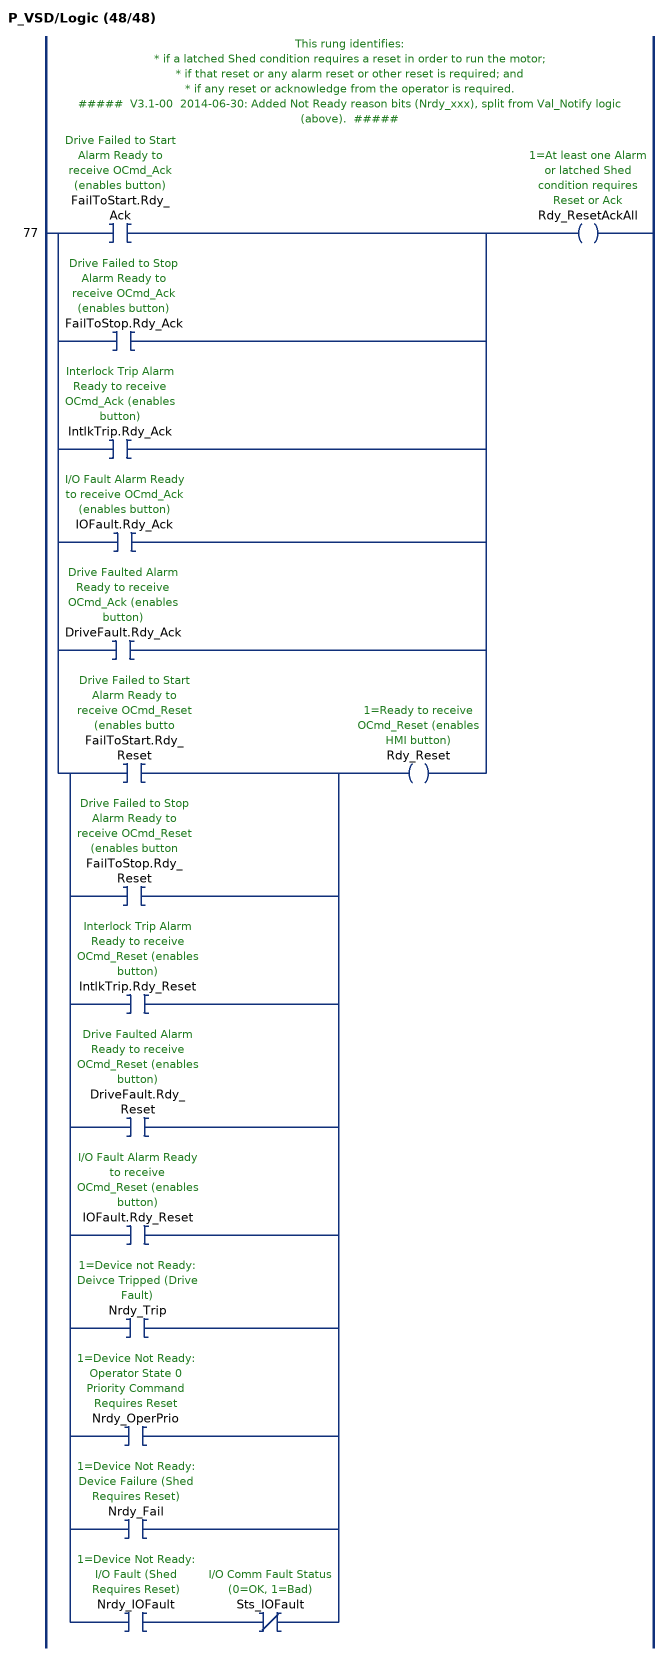
   // This rung identifies:
   // * if a latched Shed condition requires a reset in order to run the motor;
   // * if that reset or any alarm reset or other reset is required; and
   // * if any reset or acknowledge from the operator is required.
   // #####  V3.1-00  2014-06-30: Added Not Ready reason bits (Nrdy_xxx), split from Val_Notify logic (above).  #####
   77: [[XIC(FailToStart.Rdy_Ack) ,XIC(FailToStop.Rdy_Ack) ,XIC(IntlkTrip.Rdy_Ack) ,XIC(IOFault.Rdy_Ack) ,XIC(DriveFault.Rdy_Ack) ] ,[XIC(FailToStart.Rdy_Reset) ,XIC(FailToStop.Rdy_Reset) ,XIC(IntlkTrip.Rdy_Reset) ,XIC(DriveFault.Rdy_Reset) ,XIC(IOFault.Rdy_Reset) ,XIC(Nrdy_Trip) ,XIC(Nrdy_OperPrio) ,XIC(Nrdy_Fail) ,XIC(Nrdy_IOFault) XIO(Sts_IOFault) ] OTE(Rdy_Reset) ]OTE(Rdy_ResetAckAll);
END_ROUTINE

ROUTINE Prescan   (* ladder *)
// Clear Ownership, set drive to STOP, clear "lurking" Commands
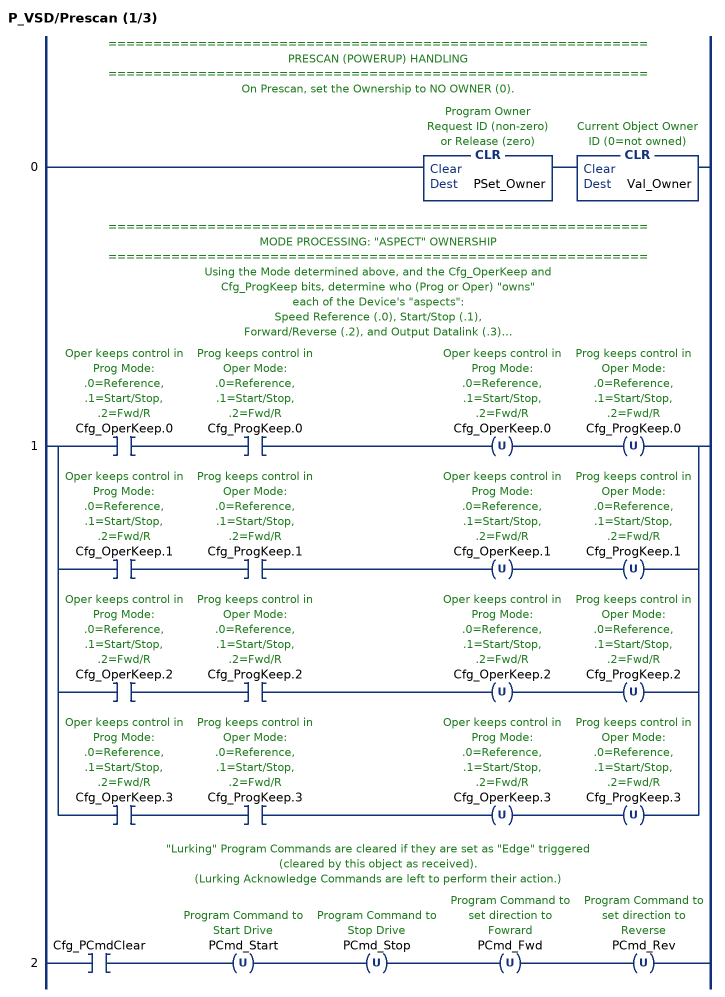
   // ============================================================
   // PRESCAN (POWERUP) HANDLING
   // ============================================================
   // On Prescan, set the Ownership to NO OWNER (0).
   0: CLR(PSet_Owner)CLR(Val_Owner);
   // ============================================================
   // MODE PROCESSING: "ASPECT" OWNERSHIP
   // ============================================================
   // Using the Mode determined above, and the Cfg_OperKeep and
   // Cfg_ProgKeep bits, determine who (Prog or Oper) "owns"
   // each of the Device's "aspects":
   // Speed Reference (.0), Start/Stop (.1),
   // Forward/Reverse (.2), and Output Datalink (.3).
   // The bits within Cfg_OperKeep and Cfg_ProgKeep determine which "aspects"
   // (sub-functions of this AOI) are retained by the Operator in Program Mode,
   // or by the Program in Operator Mode (respectively).
   // All aspects (functions) may be "kept" (basically locking the Operator/Program Mode
   // selection, rendering it moot --  you get to explain how it works to your operators!!!),
   // but it is NOT allowed to have any given function retained by BOTH Operator and
   // Program.  This rung ensures that no function is "kept" by both Oper and Prog.
   // ON PRESCAN:  If both Oper Keep and Prog Keep get set on download or during
   // controller PROG mode, they are BOTH CLEARED on powerup!!!
   // #####  V3.1-05  2016-01-22:  New rung in Prescan logic.  #####
   1: [XIC(Cfg_OperKeep.0) XIC(Cfg_ProgKeep.0) OTU(Cfg_OperKeep.0) OTU(Cfg_ProgKeep.0) ,XIC(Cfg_OperKeep.1) XIC(Cfg_ProgKeep.1) OTU(Cfg_OperKeep.1) OTU(Cfg_ProgKeep.1) ,XIC(Cfg_OperKeep.2) XIC(Cfg_ProgKeep.2) OTU(Cfg_OperKeep.2) OTU(Cfg_ProgKeep.2) ,XIC(Cfg_OperKeep.3) XIC(Cfg_ProgKeep.3) OTU(Cfg_OperKeep.3) OTU(Cfg_ProgKeep.3) ];
   // "Lurking" Program Commands are cleared if they are set as "Edge" triggered
   // (cleared by this object as received).
   // (Lurking Acknowledge Commands are left to perform their action.)
   2: XIC(Cfg_PCmdClear)OTU(PCmd_Start)OTU(PCmd_Stop)OTU(PCmd_Fwd)OTU(PCmd_Rev);
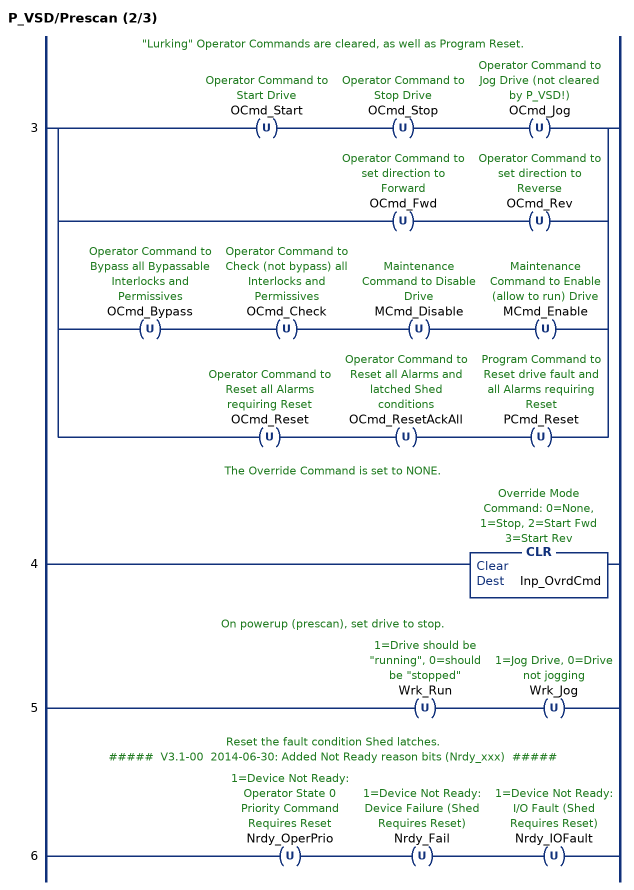
   // "Lurking" Operator Commands are cleared, as well as Program Reset.
   3: [OTU(OCmd_Start) OTU(OCmd_Stop) OTU(OCmd_Jog) ,OTU(OCmd_Fwd) OTU(OCmd_Rev) ,OTU(OCmd_Bypass) OTU(OCmd_Check) OTU(MCmd_Disable) OTU(MCmd_Enable) ,OTU(OCmd_Reset) OTU(OCmd_ResetAckAll) OTU(PCmd_Reset) ];
   // The Override Command is set to NONE.
   4: CLR(Inp_OvrdCmd);
   // On powerup (prescan), set drive to stop.
   5: OTU(Wrk_Run)OTU(Wrk_Jog);
   // Reset the fault condition Shed latches.
   // #####  V3.1-00  2014-06-30: Added Not Ready reason bits (Nrdy_xxx)  #####
   6: OTU(Nrdy_OperPrio)OTU(Nrdy_Fail)OTU(Nrdy_IOFault);
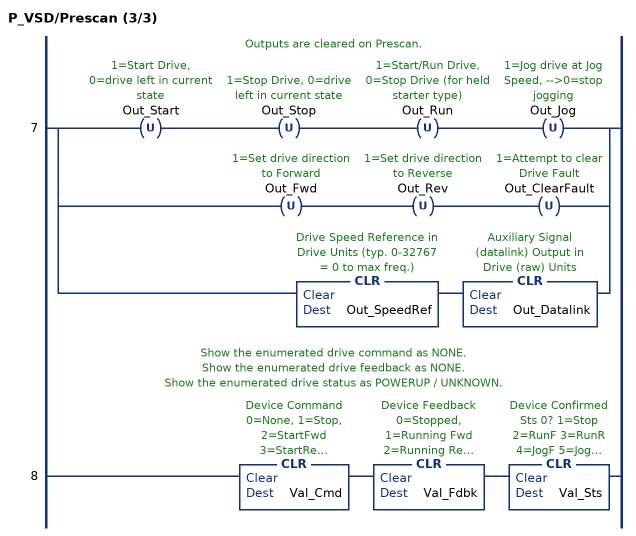
   // Outputs are cleared on Prescan.
   7: [OTU(Out_Start) OTU(Out_Stop) OTU(Out_Run) OTU(Out_Jog) ,OTU(Out_Fwd) OTU(Out_Rev) OTU(Out_ClearFault) ,CLR(Out_SpeedRef) CLR(Out_Datalink) ];
   // Show the enumerated drive command as NONE.
   // Show the enumerated drive feedback as NONE.
   // Show the enumerated drive status as POWERUP / UNKNOWN.
   8: CLR(Val_Cmd)CLR(Val_Fdbk)CLR(Val_Sts);
END_ROUTINE
END_ADD_ON_INSTRUCTION

VAR_GLOBAL   (* controller tags *)
   COCCION_TK_200 : TIMER := (PRE := 60000);
   COCCION_TK_200_LUPULO : TIMER := (PRE := 60000);
   Cond1_Nivel_TK_200 : BOOL;
   Cond2_Nivel_TK_200 : BOOL;
   Cond3_Nivel_TK_200 : BOOL;
   E0_Calentar_TK_200 : SFC_STEP := (Status := 16#0020_0000, PauseTimer := 1);
   E0_Llenar : SFC_STEP := (Status := 16#a820_0201, X := 1, SA := 1, DN := 1, PauseTimer := 1, T := 1273999, TMax := 1273999, Count := 1);
   E0_Llenar_TK_100 : SFC_STEP := (Status := 16#0020_0000, PauseTimer := 1);
   E0_Llenar_TK_200 : SFC_STEP := (Status := 16#0020_0000, PauseTimer := 1);
   E0_Moler_TK_300 : SFC_STEP := (Status := 16#0020_0000, PauseTimer := 1);
   E0_Tostado_TK_200 : SFC_STEP := (Status := 16#0020_0000, PauseTimer := 1);
   E0_Vaciado_TK_200 : SFC_STEP := (Status := 16#0020_0000, PauseTimer := 1);
   E0_Vaciado_TK_300 : SFC_STEP := (Status := 16#0020_0000, PauseTimer := 1);
   E1_Calentar_TK_200 : SFC_STEP := (Status := 16#0020_0000, PauseTimer := 1);
   E1_LLenar : SFC_STEP := (Status := 16#0020_0001, PauseTimer := 1);
   E1_LLenar_TK_100 : SFC_STEP := (Status := 16#0020_0000, PauseTimer := 1);
   E1_LLenar_TK_200 : SFC_STEP := (Status := 16#0020_0000, PauseTimer := 1);
   E1_LLenar_TK_300 : SFC_STEP := (Status := 16#0020_0000, PauseTimer := 1);
   E1_Vaciado_TK_200 : SFC_STEP := (Status := 16#0020_0000, PauseTimer := 1);
   E1_Vaciado_TK_300 : SFC_STEP := (Status := 16#0020_0000, PauseTimer := 1);
   E2_Agitar_TK_200 : SFC_STEP := (Status := 16#0020_0000, PauseTimer := 1);
   E2_Llenado_TK_100 : SFC_STEP := (Status := 16#0020_0001, PauseTimer := 1);
   E2_Llenado_TK_200 : SFC_STEP := (Status := 16#0020_0000, PauseTimer := 1);
   E2_Trirurado_TK_100 : SFC_STEP := (Status := 16#0020_0000, PauseTimer := 1);
   E3_Calentar_TK_300 : SFC_STEP := (Status := 16#0020_0000, PauseTimer := 1);
   E4_Moler_TK_300 : SFC_STEP := (Status := 16#0020_0000, PauseTimer := 1);
   FSL_200 : P_DIn := (Inp_PV := 1, Inp_Target := 1, Inp_Gate := 1, Cfg_NormTextVis := 1, Cfg_PCmdClear := 1, Cfg_TgtDisagreeAckReqd := 1, Cfg_TgtDisagreeSeverity := 750, Ack_TgtDisagree := 1);
   FV_001 : P_ValveSO := (Inp_PermOK := 1, Inp_NBPermOK := 1, Inp_IntlkOK := 1, Inp_NBIntlkOK := 1, Cfg_LSFail := 1, Cfg_PCmdClear := 1, Cfg_ProgDefault := 1, Cfg_ShedOnFullStall := 1, Cfg_ShedOnTransitStall := 1, Cfg_ShedOnIOFault := 1, Cfg_FullStallAckReqd := 1, Cfg_TransitStallAckReqd := 1, Cfg_IntlkTripAckReqd := 1, Cfg_IOFaultAckReqd := 1, Cfg_FullStallSeverity := 1000, Cfg_TransitStallSeverity := 1000, Cfg_IntlkTripSeverity := 500, Cfg_IOFaultSeverity := 1000, Cfg_SimFdbkT := 2, Cfg_FullStallT := 5, Cfg_TransitStallT := 10, Ack_FullStall := 1, Ack_TransitStall := 1, Ack_IntlkTrip := 1, Ack_IOFault := 1);
   FV_001_Intlk : P_Intlk := (Cfg_PCmdClear := 1, Sts_IntlkOK := 1, Sts_NBIntlkOK := 1);
   FV_001_Intlk1 : P_Intlk := (Cfg_PCmdClear := 1, Sts_IntlkOK := 1, Sts_NBIntlkOK := 1);
   FV_001_Perm : P_Perm := (Inp_Perm01 := 1, Inp_Perm02 := 1, Inp_Perm03 := 1, Inp_Perm04 := 1, Inp_Perm05 := 1, Inp_Perm06 := 1, Inp_Perm07 := 1, Inp_Perm08 := 1, Inp_Perm09 := 1, Inp_Perm10 := 1, Inp_Perm11 := 1, Inp_Perm12 := 1, Inp_Perm13 := 1, Inp_Perm14 := 1, Inp_Perm15 := 1, Cfg_OKState := 2#1111_1111_1111_1111, Sts_Perm := 2#1111_1111_1111_1110);
   FV_001_Perm1 : P_Perm := (Inp_Perm00 := 1, Inp_Perm01 := 1, Inp_Perm02 := 1, Inp_Perm03 := 1, Inp_Perm04 := 1, Inp_Perm05 := 1, Inp_Perm06 := 1, Inp_Perm07 := 1, Inp_Perm08 := 1, Inp_Perm09 := 1, Inp_Perm10 := 1, Inp_Perm11 := 1, Inp_Perm12 := 1, Inp_Perm13 := 1, Inp_Perm14 := 1, Inp_Perm15 := 1, Cfg_OKState := 2#1111_1111_1111_1111, Sts_PermOK := 1, Sts_NBPermOK := 1, Sts_Perm := 2#1111_1111_1111_1111);
   FV_002 : P_ValveSO := (Inp_PermOK := 1, Inp_NBPermOK := 1, Inp_IntlkOK := 1, Inp_NBIntlkOK := 1, Cfg_LSFail := 1, Cfg_PCmdClear := 1, Cfg_ProgDefault := 1, Cfg_ShedOnFullStall := 1, Cfg_ShedOnTransitStall := 1, Cfg_ShedOnIOFault := 1, Cfg_FullStallAckReqd := 1, Cfg_TransitStallAckReqd := 1, Cfg_IntlkTripAckReqd := 1, Cfg_IOFaultAckReqd := 1, Cfg_FullStallSeverity := 1000, Cfg_TransitStallSeverity := 1000, Cfg_IntlkTripSeverity := 500, Cfg_IOFaultSeverity := 1000, Cfg_SimFdbkT := 2, Cfg_FullStallT := 5, Cfg_TransitStallT := 10, Ack_FullStall := 1, Ack_TransitStall := 1, Ack_IntlkTrip := 1, Ack_IOFault := 1);
   FV_002_Intlk : P_Intlk := (Cfg_PCmdClear := 1, Sts_IntlkOK := 1, Sts_NBIntlkOK := 1);
   FV_002_Perm : P_Perm := (Inp_Perm01 := 1, Inp_Perm02 := 1, Inp_Perm03 := 1, Inp_Perm04 := 1, Inp_Perm05 := 1, Inp_Perm06 := 1, Inp_Perm07 := 1, Inp_Perm08 := 1, Inp_Perm09 := 1, Inp_Perm10 := 1, Inp_Perm11 := 1, Inp_Perm12 := 1, Inp_Perm13 := 1, Inp_Perm14 := 1, Inp_Perm15 := 1, Cfg_OKState := 2#1111_1111_1111_1111, Sts_Perm := 2#1111_1111_1111_1110);
   FV_003 : P_ValveSO := (Inp_PermOK := 1, Inp_NBPermOK := 1, Inp_IntlkOK := 1, Inp_NBIntlkOK := 1, Cfg_LSFail := 1, Cfg_PCmdClear := 1, Cfg_ProgDefault := 1, Cfg_ShedOnFullStall := 1, Cfg_ShedOnTransitStall := 1, Cfg_ShedOnIOFault := 1, Cfg_FullStallAckReqd := 1, Cfg_TransitStallAckReqd := 1, Cfg_IntlkTripAckReqd := 1, Cfg_IOFaultAckReqd := 1, Cfg_FullStallSeverity := 1000, Cfg_TransitStallSeverity := 1000, Cfg_IntlkTripSeverity := 500, Cfg_IOFaultSeverity := 1000, Cfg_SimFdbkT := 2, Cfg_FullStallT := 5, Cfg_TransitStallT := 10, Ack_FullStall := 1, Ack_TransitStall := 1, Ack_IntlkTrip := 1, Ack_IOFault := 1);
   FV_003_Perm : P_Perm := (Inp_Perm00 := 1, Inp_Perm01 := 1, Inp_Perm02 := 1, Inp_Perm03 := 1, Inp_Perm04 := 1, Inp_Perm05 := 1, Inp_Perm06 := 1, Inp_Perm07 := 1, Inp_Perm08 := 1, Inp_Perm09 := 1, Inp_Perm10 := 1, Inp_Perm11 := 1, Inp_Perm12 := 1, Inp_Perm13 := 1, Inp_Perm14 := 1, Inp_Perm15 := 1, Cfg_OKState := 2#1111_1111_1111_1111, Sts_PermOK := 1, Sts_NBPermOK := 1, Sts_Perm := 2#1111_1111_1111_1111);
   FV_003_Perm1_ok : BOOL;
   FV_003_Perm_ok : BOOL;
   FV_004 : P_ValveSO := (Inp_PermOK := 1, Inp_NBPermOK := 1, Inp_IntlkOK := 1, Inp_NBIntlkOK := 1, Cfg_LSFail := 1, Cfg_PCmdClear := 1, Cfg_ProgDefault := 1, Cfg_ShedOnFullStall := 1, Cfg_ShedOnTransitStall := 1, Cfg_ShedOnIOFault := 1, Cfg_FullStallAckReqd := 1, Cfg_TransitStallAckReqd := 1, Cfg_IntlkTripAckReqd := 1, Cfg_IOFaultAckReqd := 1, Cfg_FullStallSeverity := 1000, Cfg_TransitStallSeverity := 1000, Cfg_IntlkTripSeverity := 500, Cfg_IOFaultSeverity := 1000, Cfg_SimFdbkT := 2, Cfg_FullStallT := 5, Cfg_TransitStallT := 10, Ack_FullStall := 1, Ack_TransitStall := 1, Ack_IntlkTrip := 1, Ack_IOFault := 1);
   FV_005 : P_ValveSO := (Inp_PermOK := 1, Inp_NBPermOK := 1, Inp_IntlkOK := 1, Inp_NBIntlkOK := 1, Cfg_LSFail := 1, Cfg_PCmdClear := 1, Cfg_ProgDefault := 1, Cfg_ShedOnFullStall := 1, Cfg_ShedOnTransitStall := 1, Cfg_ShedOnIOFault := 1, Cfg_FullStallAckReqd := 1, Cfg_TransitStallAckReqd := 1, Cfg_IntlkTripAckReqd := 1, Cfg_IOFaultAckReqd := 1, Cfg_FullStallSeverity := 1000, Cfg_TransitStallSeverity := 1000, Cfg_IntlkTripSeverity := 500, Cfg_IOFaultSeverity := 1000, Cfg_SimFdbkT := 2, Cfg_FullStallT := 5, Cfg_TransitStallT := 10, Ack_FullStall := 1, Ack_TransitStall := 1, Ack_IntlkTrip := 1, Ack_IOFault := 1);
   FV_006 : P_ValveSO := (Inp_PermOK := 1, Inp_NBPermOK := 1, Inp_IntlkOK := 1, Inp_NBIntlkOK := 1, Cfg_LSFail := 1, Cfg_PCmdClear := 1, Cfg_ShedOnFullStall := 1, Cfg_ShedOnTransitStall := 1, Cfg_ShedOnIOFault := 1, Cfg_FullStallAckReqd := 1, Cfg_TransitStallAckReqd := 1, Cfg_IntlkTripAckReqd := 1, Cfg_IOFaultAckReqd := 1, Cfg_FullStallSeverity := 1000, Cfg_TransitStallSeverity := 1000, Cfg_IntlkTripSeverity := 500, Cfg_IOFaultSeverity := 1000, Cfg_SimFdbkT := 2, Cfg_FullStallT := 5, Cfg_TransitStallT := 10, Ack_FullStall := 1, Ack_TransitStall := 1, Ack_IntlkTrip := 1, Ack_IOFault := 1);
   FV_00_Intlk_Ok : BOOL;
   FV_00_Perm_Ok : BOOL;
   FV_100 : P_ValveSO := (Inp_PermOK := 1, Inp_NBPermOK := 1, Inp_IntlkOK := 1, Inp_NBIntlkOK := 1, Cfg_LSFail := 1, Cfg_PCmdClear := 1, Cfg_ProgDefault := 1, Cfg_ShedOnFullStall := 1, Cfg_ShedOnTransitStall := 1, Cfg_ShedOnIOFault := 1, Cfg_FullStallAckReqd := 1, Cfg_TransitStallAckReqd := 1, Cfg_IntlkTripAckReqd := 1, Cfg_IOFaultAckReqd := 1, Cfg_FullStallSeverity := 1000, Cfg_TransitStallSeverity := 1000, Cfg_IntlkTripSeverity := 500, Cfg_IOFaultSeverity := 1000, Cfg_SimFdbkT := 2, Cfg_FullStallT := 5, Cfg_TransitStallT := 10, Ack_FullStall := 1, Ack_TransitStall := 1, Ack_IntlkTrip := 1, Ack_IOFault := 1);
   FV_100_Intlk : P_Intlk := (Cfg_PCmdClear := 1, Sts_IntlkOK := 1, Sts_NBIntlkOK := 1);
   FV_100_Intlk1 : P_Intlk := (Cfg_PCmdClear := 1, Sts_IntlkOK := 1, Sts_NBIntlkOK := 1);
   FV_100_Perm : P_Perm := (Inp_Perm00 := 1, Inp_Perm01 := 1, Inp_Perm02 := 1, Inp_Perm03 := 1, Inp_Perm04 := 1, Inp_Perm05 := 1, Inp_Perm06 := 1, Inp_Perm07 := 1, Inp_Perm08 := 1, Inp_Perm09 := 1, Inp_Perm10 := 1, Inp_Perm11 := 1, Inp_Perm12 := 1, Inp_Perm13 := 1, Inp_Perm14 := 1, Inp_Perm15 := 1, Cfg_OKState := 2#1111_1111_1111_1111, Sts_PermOK := 1, Sts_NBPermOK := 1, Sts_Perm := 2#1111_1111_1111_1111);
   FV_100_Perm1 : P_Perm := (Inp_Perm00 := 1, Inp_Perm01 := 1, Inp_Perm02 := 1, Inp_Perm03 := 1, Inp_Perm04 := 1, Inp_Perm05 := 1, Inp_Perm06 := 1, Inp_Perm07 := 1, Inp_Perm08 := 1, Inp_Perm09 := 1, Inp_Perm10 := 1, Inp_Perm11 := 1, Inp_Perm12 := 1, Inp_Perm13 := 1, Inp_Perm14 := 1, Inp_Perm15 := 1, Cfg_OKState := 2#1111_1111_1111_1111, Sts_PermOK := 1, Sts_NBPermOK := 1, Sts_Perm := 2#1111_1111_1111_1111);
   INTLK_OK_P_51_AB : BOOL;
   LIT_100 : P_AIn := (Inp_PV := 3277.0, Inp_HiHiGate := 1, Inp_HiGate := 1, Inp_LoGate := 1, Inp_LoLoGate := 1, Inp_FailGate := 1, Cfg_SetTrack := 1, Cfg_PCmdClear := 1, Cfg_HiHiAckReqd := 1, Cfg_HiAckReqd := 1, Cfg_LoAckReqd := 1, Cfg_LoLoAckReqd := 1, Cfg_FailAckReqd := 1, Cfg_HiHiSeverity := 750, Cfg_HiSeverity := 500, Cfg_LoSeverity := 500, Cfg_LoLoSeverity := 750, Cfg_FailSeverity := 1000, Cfg_InpRawMin := 3277.0, Cfg_InpRawMax := 16384.0, Cfg_PVEUMax := 4000.0, Cfg_HiHiDB := 1.0, Cfg_HiDB := 1.0, Cfg_LoDB := 1.0, Cfg_LoLoDB := 1.0, Cfg_FailHiLim := 4000.0, Cfg_FailLoLim := -2.0833333, Cfg_FailDB := 0.41666666, PSet_HiHiLim := 4000.0, PSet_HiLim := 3900.0, OSet_HiHiLim := 4000.0, OSet_HiLim := 3900.0, Val_PVEUMax := 4000.0, SrcQ_IO := 1, SrcQ := 1, Val_Fault := 24, Val_Mode := 9, Val_HiHiLim := 90.0, Val_HiLim := 80.0, Sts_InpPV := 1, Sts_Oper := 1, Sts_HiHiGate := 1, Ack_HiHi := 1, Sts_HiGate := 1, Ack_Hi := 1, Sts_LoCmp := 1, Sts_LoGate := 1, Sts_Lo := 1, Ack_Lo := 1, Sts_LoLoCmp := 1, Sts_LoLoGate := 1, Sts_LoLo := 1, Ack_LoLo := 1, Sts_FailGate := 1, Ack_Fail := 1, Rdy_OSet := 1);
   LIT_101 : P_AIn := (Inp_PV := 3277.0, Inp_HiHiGate := 1, Inp_HiGate := 1, Inp_LoGate := 1, Inp_LoLoGate := 1, Inp_FailGate := 1, Cfg_SetTrack := 1, Cfg_PCmdClear := 1, Cfg_HiHiAckReqd := 1, Cfg_HiAckReqd := 1, Cfg_LoAckReqd := 1, Cfg_LoLoAckReqd := 1, Cfg_FailAckReqd := 1, Cfg_HiHiSeverity := 750, Cfg_HiSeverity := 500, Cfg_LoSeverity := 500, Cfg_LoLoSeverity := 750, Cfg_FailSeverity := 1000, Cfg_InpRawMin := 3277.0, Cfg_InpRawMax := 16384.0, Cfg_PVEUMax := 4000.0, Cfg_HiHiDB := 1.0, Cfg_HiDB := 1.0, Cfg_LoDB := 1.0, Cfg_LoLoDB := 1.0, Cfg_FailHiLim := 103.958336, Cfg_FailLoLim := -2.0833333, Cfg_FailDB := 0.41666666, PSet_HiHiLim := 90.0, PSet_HiLim := 80.0, OSet_HiHiLim := 90.0, OSet_HiLim := 80.0, Val_PVEUMax := 4000.0, SrcQ_IO := 1, SrcQ := 1, Val_Fault := 24, Val_Mode := 9, Val_HiHiLim := 90.0, Val_HiLim := 80.0, Sts_InpPV := 1, Sts_Oper := 1, Sts_HiHiGate := 1, Ack_HiHi := 1, Sts_HiGate := 1, Ack_Hi := 1, Sts_LoCmp := 1, Sts_LoGate := 1, Sts_Lo := 1, Ack_Lo := 1, Sts_LoLoCmp := 1, Sts_LoLoGate := 1, Sts_LoLo := 1, Ack_LoLo := 1, Sts_FailGate := 1, Ack_Fail := 1, Rdy_OSet := 1);
   LIT_102 : P_AIn := (Inp_PV := 3277.0, Inp_HiHiGate := 1, Inp_HiGate := 1, Inp_LoGate := 1, Inp_LoLoGate := 1, Inp_FailGate := 1, Cfg_SetTrack := 1, Cfg_PCmdClear := 1, Cfg_HiHiAckReqd := 1, Cfg_HiAckReqd := 1, Cfg_LoAckReqd := 1, Cfg_LoLoAckReqd := 1, Cfg_FailAckReqd := 1, Cfg_HiHiSeverity := 750, Cfg_HiSeverity := 500, Cfg_LoSeverity := 500, Cfg_LoLoSeverity := 750, Cfg_FailSeverity := 1000, Cfg_InpRawMin := 3277.0, Cfg_InpRawMax := 16384.0, Cfg_PVEUMax := 4000.0, Cfg_HiHiDB := 1.0, Cfg_HiDB := 1.0, Cfg_LoDB := 1.0, Cfg_LoLoDB := 1.0, Cfg_FailHiLim := 103.958336, Cfg_FailLoLim := -2.0833333, Cfg_FailDB := 0.41666666, PSet_HiHiLim := 90.0, PSet_HiLim := 80.0, OSet_HiHiLim := 90.0, OSet_HiLim := 80.0, Val_PVEUMax := 4000.0, SrcQ_IO := 1, SrcQ := 1, Val_Fault := 24, Val_Mode := 9, Val_HiHiLim := 90.0, Val_HiLim := 80.0, Sts_InpPV := 1, Sts_Oper := 1, Sts_HiHiGate := 1, Ack_HiHi := 1, Sts_HiGate := 1, Ack_Hi := 1, Sts_LoCmp := 1, Sts_LoGate := 1, Sts_Lo := 1, Ack_Lo := 1, Sts_LoLoCmp := 1, Sts_LoLoGate := 1, Sts_LoLo := 1, Ack_LoLo := 1, Sts_FailGate := 1, Ack_Fail := 1, Rdy_OSet := 1);
   LIT_200 : P_AIn := (Inp_HiHiGate := 1, Inp_HiGate := 1, Inp_LoGate := 1, Inp_LoLoGate := 1, Inp_FailGate := 1, Cfg_SetTrack := 1, Cfg_PCmdClear := 1, Cfg_ProgDefault := 1, Cfg_HiHiAckReqd := 1, Cfg_HiAckReqd := 1, Cfg_LoAckReqd := 1, Cfg_LoLoAckReqd := 1, Cfg_FailAckReqd := 1, Cfg_HiHiSeverity := 750, Cfg_HiSeverity := 500, Cfg_LoSeverity := 500, Cfg_LoLoSeverity := 750, Cfg_FailSeverity := 1000, Cfg_InpRawMin := 3277.0, Cfg_InpRawMax := 16384.0, Cfg_PVEUMax := 100.0, Cfg_HiHiDB := 1.0, Cfg_HiDB := 1.0, Cfg_LoDB := 1.0, Cfg_LoLoDB := 1.0, Cfg_FailHiLim := 103.958336, Cfg_FailLoLim := -2.0833333, Cfg_FailDB := 0.41666666, PSet_HiHiLim := 1.5e+38, PSet_HiLim := 1.5e+38, PSet_LoLim := -1.5e+38, PSet_LoLoLim := -1.5e+38, OSet_HiHiLim := 1.5e+38, OSet_HiLim := 1.5e+38, OSet_LoLim := -1.5e+38, OSet_LoLoLim := -1.5e+38, Val_PVMinCapt := 1.5e+38, Val_PVMaxCapt := -1.5e+38, Val_PVEUMax := 100.0, Val_HiHiLim := 1.5e+38, Val_HiLim := 1.5e+38, Val_LoLim := -1.5e+38, Val_LoLoLim := -1.5e+38, Sts_InpPV := 1, Sts_Oper := 1, Ack_HiHi := 1, Ack_Hi := 1, Ack_Lo := 1, Ack_LoLo := 1, Ack_Fail := 1);
   LLENADO_TK_200_LUPULO : TIMER := (PRE := 10000);
   Llenar_T1 : BOOL;
   Llenar_T2 : BOOL;
   Llenar_T_100 : BOOL;
   Llenar_TK_100 : BOOL;
   LSH_100 : P_DIn := (Inp_Target := 1, Inp_Gate := 1, Cfg_NormTextVis := 1, Cfg_PCmdClear := 1, Cfg_TgtDisagreeAckReqd := 1, Cfg_TgtDisagreeSeverity := 750, SrcQ_IO := 1, SrcQ := 1, Val_Fault := 16, Sts_InpPV := 1, Sts_TgtDisagreeCmp := 1, Sts_TgtDisagreeGate := 1, Sts_TgtDisagree := 1, Ack_TgtDisagree := 1, Rdy_SubstPV := 1);
   LSL_100 : P_DIn := (Inp_Target := 1, Inp_Gate := 1, Cfg_NormTextVis := 1, Cfg_PCmdClear := 1, Cfg_TgtDisagreeAckReqd := 1, Cfg_TgtDisagreeSeverity := 750, SrcQ_IO := 1, SrcQ := 1, Val_Fault := 16, Sts_PV := 1, Sts_InpPV := 1, Sts_TgtDisagreeCmp := 1, Sts_TgtDisagreeGate := 1, Sts_TgtDisagree := 1, Ack_TgtDisagree := 1, Rdy_SubstPV := 1);
   LSL_101 : P_DIn := (Inp_PV := 1, Inp_Target := 1, Inp_Gate := 1, Cfg_NormTextVis := 1, Cfg_PCmdClear := 1, Cfg_TgtDisagreeAckReqd := 1, Cfg_TgtDisagreeSeverity := 750, Ack_TgtDisagree := 1);
   LSL_201 : P_DIn := (Inp_PV := 1, Inp_Target := 1, Inp_Gate := 1, Cfg_NormTextVis := 1, Cfg_PCmdClear := 1, Cfg_TgtDisagreeAckReqd := 1, Cfg_TgtDisagreeSeverity := 750, Ack_TgtDisagree := 1);
   LSL_202 : P_DIn := (Inp_PV := 1, Inp_Target := 1, Inp_Gate := 1, Cfg_NormTextVis := 1, Cfg_PCmdClear := 1, Cfg_TgtDisagreeAckReqd := 1, Cfg_TgtDisagreeSeverity := 750, Ack_TgtDisagree := 1);
   LZT_52 : P_AIn := (Inp_HiHiGate := 1, Inp_HiGate := 1, Inp_LoGate := 1, Inp_LoLoGate := 1, Inp_FailGate := 1, Cfg_SetTrack := 1, Cfg_PCmdClear := 1, Cfg_ProgDefault := 1, Cfg_HiHiAckReqd := 1, Cfg_HiAckReqd := 1, Cfg_LoAckReqd := 1, Cfg_LoLoAckReqd := 1, Cfg_FailAckReqd := 1, Cfg_HiHiSeverity := 750, Cfg_HiSeverity := 500, Cfg_LoSeverity := 500, Cfg_LoLoSeverity := 750, Cfg_FailSeverity := 1000, Cfg_InpRawMin := 3277.0, Cfg_InpRawMax := 16384.0, Cfg_PVEUMax := 100.0, Cfg_HiHiDB := 1.0, Cfg_HiDB := 1.0, Cfg_LoDB := 1.0, Cfg_LoLoDB := 1.0, Cfg_FailHiLim := 103.958336, Cfg_FailLoLim := -2.0833333, Cfg_FailDB := 0.41666666, PSet_HiHiLim := 1.5e+38, PSet_HiLim := 1.5e+38, PSet_LoLim := -1.5e+38, PSet_LoLoLim := -1.5e+38, OSet_HiHiLim := 1.5e+38, OSet_HiLim := 1.5e+38, OSet_LoLim := -1.5e+38, OSet_LoLoLim := -1.5e+38, Val_PVMinCapt := 1.5e+38, Val_PVMaxCapt := -1.5e+38, Val_PVEUMax := 100.0, Val_HiHiLim := 1.5e+38, Val_HiLim := 1.5e+38, Val_LoLim := -1.5e+38, Val_LoLoLim := -1.5e+38, Sts_InpPV := 1, Sts_Oper := 1, Ack_HiHi := 1, Ack_Hi := 1, Ack_Lo := 1, Ack_LoLo := 1, Ack_Fail := 1);
   M_001 : P_Motor := (Inp_PermOK := 1, Inp_NBPermOK := 1, Inp_IntlkOK := 1, Inp_NBIntlkOK := 1, Cfg_PCmdClear := 1, Cfg_ProgDefault := 1, Cfg_ShedOnFailToStart := 1, Cfg_ShedOnIOFault := 1, Cfg_FailToStartAckReqd := 1, Cfg_FailToStopAckReqd := 1, Cfg_IntlkTripAckReqd := 1, Cfg_IOFaultAckReqd := 1, Cfg_FailToStartSeverity := 1000, Cfg_FailToStopSeverity := 1000, Cfg_IntlkTripSeverity := 500, Cfg_IOFaultSeverity := 1000, Cfg_SimFdbkT := 2, Cfg_FailToStartT := 10, Cfg_FailToStopT := 10, Sts_Stopped := 1, Sts_Oper := 1, Ack_FailToStart := 1, Ack_FailToStop := 1, Ack_IntlkTrip := 1, Ack_IOFault := 1);
   M_001_Intlk : P_Intlk := (Cfg_PCmdClear := 1, Sts_IntlkOK := 1, Sts_NBIntlkOK := 1);
   M_001_Perm : P_Perm := (Inp_Perm02 := 1, Inp_Perm03 := 1, Inp_Perm04 := 1, Inp_Perm05 := 1, Inp_Perm06 := 1, Inp_Perm07 := 1, Inp_Perm08 := 1, Inp_Perm09 := 1, Inp_Perm10 := 1, Inp_Perm11 := 1, Inp_Perm12 := 1, Inp_Perm13 := 1, Inp_Perm14 := 1, Inp_Perm15 := 1, Cfg_OKState := 2#1111_1111_1111_1111, Sts_Perm := 2#1111_1111_1111_1100);
   M_100 : P_VSD := (Inp_Ready := 1, Inp_CommandDir := 1, Inp_ActualDir := 1, Inp_FwdPermOK := 1, Inp_FwdNBPermOK := 1, Inp_RevPermOK := 1, Inp_RevNBPermOK := 1, Inp_IntlkOK := 1, Inp_NBIntlkOK := 1, Cfg_SetTrack := 1, Cfg_PCmdClear := 1, Cfg_ProgDefault := 1, Cfg_ShedOnFailToStart := 1, Cfg_ShedOnIOFault := 1, Cfg_FailToStartAckReqd := 1, Cfg_FailToStopAckReqd := 1, Cfg_IntlkTripAckReqd := 1, Cfg_DriveFaultAckReqd := 1, Cfg_IOFaultAckReqd := 1, Cfg_FailToStartSeverity := 1000, Cfg_FailToStopSeverity := 1000, Cfg_IntlkTripSeverity := 500, Cfg_DriveFaultSeverity := 1000, Cfg_IOFaultSeverity := 1000, Cfg_MaxSpdRef := 60.0, Cfg_SpeedRefRawMax := 32767.0, Cfg_SpeedRefEUMax := 130.0, Cfg_SpeedFdbkRawMax := 32767.0, Cfg_SpeedFdbkEUMax := 130.0, Cfg_InpDatalinkRawMax := 4095.0, Cfg_InpDatalinkEUMax := 409.5, Cfg_OutDatalinkMax := 100.0, Cfg_OutDatalinkRawMax := 4095.0, Cfg_OutDatalinkEUMax := 409.5, Cfg_SimRampT := 10, Cfg_FailToStartT := 15, Cfg_FailToStopT := 15, Cfg_ResetPulseT := 2, Val_SpeedRefEUMax := 130.0, Val_SpeedFdbkEUMax := 130.0, Ack_FailToStart := 1, Ack_FailToStop := 1, Ack_IntlkTrip := 1, Ack_DriveFault := 1, Ack_IOFault := 1);
   M_200 : P_VSD := (Inp_Ready := 1, Inp_CommandDir := 1, Inp_ActualDir := 1, Inp_FwdPermOK := 1, Inp_FwdNBPermOK := 1, Inp_RevPermOK := 1, Inp_RevNBPermOK := 1, Inp_IntlkOK := 1, Inp_NBIntlkOK := 1, Cfg_SetTrack := 1, Cfg_PCmdClear := 1, Cfg_ProgDefault := 1, Cfg_ShedOnFailToStart := 1, Cfg_ShedOnIOFault := 1, Cfg_FailToStartAckReqd := 1, Cfg_FailToStopAckReqd := 1, Cfg_IntlkTripAckReqd := 1, Cfg_DriveFaultAckReqd := 1, Cfg_IOFaultAckReqd := 1, Cfg_FailToStartSeverity := 1000, Cfg_FailToStopSeverity := 1000, Cfg_IntlkTripSeverity := 500, Cfg_DriveFaultSeverity := 1000, Cfg_IOFaultSeverity := 1000, Cfg_MaxSpdRef := 60.0, Cfg_SpeedRefRawMax := 32767.0, Cfg_SpeedRefEUMax := 130.0, Cfg_SpeedFdbkRawMax := 32767.0, Cfg_SpeedFdbkEUMax := 130.0, Cfg_InpDatalinkRawMax := 4095.0, Cfg_InpDatalinkEUMax := 409.5, Cfg_OutDatalinkMax := 100.0, Cfg_OutDatalinkRawMax := 4095.0, Cfg_OutDatalinkEUMax := 409.5, Cfg_SimRampT := 10, Cfg_FailToStartT := 15, Cfg_FailToStopT := 15, Cfg_ResetPulseT := 2, Val_SpeedRefEUMax := 130.0, Val_SpeedFdbkEUMax := 130.0, Ack_FailToStart := 1, Ack_FailToStop := 1, Ack_IntlkTrip := 1, Ack_DriveFault := 1, Ack_IOFault := 1);
   M_300 : P_VSD := (Inp_Ready := 1, Inp_CommandDir := 1, Inp_ActualDir := 1, Inp_FwdPermOK := 1, Inp_FwdNBPermOK := 1, Inp_RevPermOK := 1, Inp_RevNBPermOK := 1, Inp_IntlkOK := 1, Inp_NBIntlkOK := 1, Cfg_SetTrack := 1, Cfg_PCmdClear := 1, Cfg_ProgDefault := 1, Cfg_ShedOnFailToStart := 1, Cfg_ShedOnIOFault := 1, Cfg_FailToStartAckReqd := 1, Cfg_FailToStopAckReqd := 1, Cfg_IntlkTripAckReqd := 1, Cfg_DriveFaultAckReqd := 1, Cfg_IOFaultAckReqd := 1, Cfg_FailToStartSeverity := 1000, Cfg_FailToStopSeverity := 1000, Cfg_IntlkTripSeverity := 500, Cfg_DriveFaultSeverity := 1000, Cfg_IOFaultSeverity := 1000, Cfg_MaxSpdRef := 60.0, Cfg_SpeedRefRawMax := 32767.0, Cfg_SpeedRefEUMax := 130.0, Cfg_SpeedFdbkRawMax := 32767.0, Cfg_SpeedFdbkEUMax := 130.0, Cfg_InpDatalinkRawMax := 4095.0, Cfg_InpDatalinkEUMax := 409.5, Cfg_OutDatalinkMax := 100.0, Cfg_OutDatalinkRawMax := 4095.0, Cfg_OutDatalinkEUMax := 409.5, Cfg_SimRampT := 10, Cfg_FailToStartT := 15, Cfg_FailToStopT := 15, Cfg_ResetPulseT := 2, Val_SpeedRefEUMax := 130.0, Val_SpeedFdbkEUMax := 130.0, Ack_FailToStart := 1, Ack_FailToStop := 1, Ack_IntlkTrip := 1, Ack_DriveFault := 1, Ack_IOFault := 1);
   M_VSD_200 : P_VSD := (Inp_Ready := 1, Inp_CommandDir := 1, Inp_ActualDir := 1, Inp_FwdPermOK := 1, Inp_FwdNBPermOK := 1, Inp_RevPermOK := 1, Inp_RevNBPermOK := 1, Inp_IntlkOK := 1, Inp_NBIntlkOK := 1, Cfg_SetTrack := 1, Cfg_PCmdClear := 1, Cfg_ProgDefault := 1, Cfg_ShedOnFailToStart := 1, Cfg_ShedOnIOFault := 1, Cfg_FailToStartAckReqd := 1, Cfg_FailToStopAckReqd := 1, Cfg_IntlkTripAckReqd := 1, Cfg_DriveFaultAckReqd := 1, Cfg_IOFaultAckReqd := 1, Cfg_FailToStartSeverity := 1000, Cfg_FailToStopSeverity := 1000, Cfg_IntlkTripSeverity := 500, Cfg_DriveFaultSeverity := 1000, Cfg_IOFaultSeverity := 1000, Cfg_MaxSpdRef := 60.0, Cfg_SpeedRefRawMax := 32767.0, Cfg_SpeedRefEUMax := 130.0, Cfg_SpeedFdbkRawMax := 32767.0, Cfg_SpeedFdbkEUMax := 130.0, Cfg_InpDatalinkRawMax := 4095.0, Cfg_InpDatalinkEUMax := 409.5, Cfg_OutDatalinkMax := 100.0, Cfg_OutDatalinkRawMax := 4095.0, Cfg_OutDatalinkEUMax := 409.5, Cfg_SimRampT := 10, Cfg_FailToStartT := 15, Cfg_FailToStopT := 15, Cfg_ResetPulseT := 2, Val_SpeedRefEUMax := 130.0, Val_SpeedFdbkEUMax := 130.0, Ack_FailToStart := 1, Ack_FailToStop := 1, Ack_IntlkTrip := 1, Ack_DriveFault := 1, Ack_IOFault := 1);
   MIXER_VSD_100 : P_VSD := (Inp_Ready := 1, Inp_CommandDir := 1, Inp_ActualDir := 1, Inp_FwdPermOK := 1, Inp_FwdNBPermOK := 1, Inp_RevPermOK := 1, Inp_RevNBPermOK := 1, Inp_IntlkOK := 1, Inp_NBIntlkOK := 1, Cfg_SetTrack := 1, Cfg_PCmdClear := 1, Cfg_ProgDefault := 1, Cfg_ShedOnFailToStart := 1, Cfg_ShedOnIOFault := 1, Cfg_FailToStartAckReqd := 1, Cfg_FailToStopAckReqd := 1, Cfg_IntlkTripAckReqd := 1, Cfg_DriveFaultAckReqd := 1, Cfg_IOFaultAckReqd := 1, Cfg_FailToStartSeverity := 1000, Cfg_FailToStopSeverity := 1000, Cfg_IntlkTripSeverity := 500, Cfg_DriveFaultSeverity := 1000, Cfg_IOFaultSeverity := 1000, Cfg_MaxSpdRef := 60.0, Cfg_SpeedRefRawMax := 32767.0, Cfg_SpeedRefEUMax := 130.0, Cfg_SpeedFdbkRawMax := 32767.0, Cfg_SpeedFdbkEUMax := 130.0, Cfg_InpDatalinkRawMax := 4095.0, Cfg_InpDatalinkEUMax := 409.5, Cfg_OutDatalinkMax := 100.0, Cfg_OutDatalinkRawMax := 4095.0, Cfg_OutDatalinkEUMax := 409.5, Cfg_SimRampT := 10, Cfg_FailToStartT := 15, Cfg_FailToStopT := 15, Cfg_ResetPulseT := 2, PCmd_Stop := 1, Out_Fwd := 1, Val_SpeedRefEUMax := 130.0, Val_SpeedFdbkEUMax := 130.0, SrcQ_IO := 2, SrcQ := 2, Val_Sts := 1, Val_Mode := 9, Sts_Stopped := 1, Sts_CommandDir := 1, Sts_ActualDir := 1, Sts_Oper := 1, Ack_FailToStart := 1, Ack_FailToStop := 1, Ack_IntlkTrip := 1, Ack_DriveFault := 1, Ack_IOFault := 1, Rdy_Start := 1, Rdy_Stop := 1, Rdy_Bypass := 1, Rdy_SpeedRef := 1, Rdy_OSet := 1);
   MIXER_VSD_101 : P_VSD := (Inp_Ready := 1, Inp_CommandDir := 1, Inp_ActualDir := 1, Inp_FwdPermOK := 1, Inp_FwdNBPermOK := 1, Inp_RevPermOK := 1, Inp_RevNBPermOK := 1, Inp_IntlkOK := 1, Inp_NBIntlkOK := 1, Cfg_SetTrack := 1, Cfg_PCmdClear := 1, Cfg_ProgDefault := 1, Cfg_ShedOnFailToStart := 1, Cfg_ShedOnIOFault := 1, Cfg_FailToStartAckReqd := 1, Cfg_FailToStopAckReqd := 1, Cfg_IntlkTripAckReqd := 1, Cfg_DriveFaultAckReqd := 1, Cfg_IOFaultAckReqd := 1, Cfg_FailToStartSeverity := 1000, Cfg_FailToStopSeverity := 1000, Cfg_IntlkTripSeverity := 500, Cfg_DriveFaultSeverity := 1000, Cfg_IOFaultSeverity := 1000, Cfg_MaxSpdRef := 60.0, Cfg_SpeedRefRawMax := 32767.0, Cfg_SpeedRefEUMax := 130.0, Cfg_SpeedFdbkRawMax := 32767.0, Cfg_SpeedFdbkEUMax := 130.0, Cfg_InpDatalinkRawMax := 4095.0, Cfg_InpDatalinkEUMax := 409.5, Cfg_OutDatalinkMax := 100.0, Cfg_OutDatalinkRawMax := 4095.0, Cfg_OutDatalinkEUMax := 409.5, Cfg_SimRampT := 10, Cfg_FailToStartT := 15, Cfg_FailToStopT := 15, Cfg_ResetPulseT := 2, PCmd_Stop := 1, Out_Fwd := 1, Val_SpeedRefEUMax := 130.0, Val_SpeedFdbkEUMax := 130.0, SrcQ_IO := 2, SrcQ := 2, Val_Sts := 1, Val_Mode := 9, Sts_Stopped := 1, Sts_CommandDir := 1, Sts_ActualDir := 1, Sts_Oper := 1, Ack_FailToStart := 1, Ack_FailToStop := 1, Ack_IntlkTrip := 1, Ack_DriveFault := 1, Ack_IOFault := 1, Rdy_Start := 1, Rdy_Stop := 1, Rdy_Bypass := 1, Rdy_SpeedRef := 1, Rdy_OSet := 1);
   Motor_Intlk1_OK : BOOL;
   Motor_Intlk_OK : BOOL;
   Nivel_TK_200 : BOOL;
   NO_interlock : BOOL;   // Condiciones de seguridad no se cumplen
   ok_interlock : BOOL;   // Condiciones de seguridad no se cumplen
   P_100_B : P_VSD := (Inp_Ready := 1, Inp_CommandDir := 1, Inp_ActualDir := 1, Inp_FwdPermOK := 1, Inp_FwdNBPermOK := 1, Inp_RevPermOK := 1, Inp_RevNBPermOK := 1, Inp_IntlkOK := 1, Inp_NBIntlkOK := 1, Cfg_SetTrack := 1, Cfg_PCmdClear := 1, Cfg_ProgDefault := 1, Cfg_ShedOnFailToStart := 1, Cfg_ShedOnIOFault := 1, Cfg_FailToStartAckReqd := 1, Cfg_FailToStopAckReqd := 1, Cfg_IntlkTripAckReqd := 1, Cfg_DriveFaultAckReqd := 1, Cfg_IOFaultAckReqd := 1, Cfg_FailToStartSeverity := 1000, Cfg_FailToStopSeverity := 1000, Cfg_IntlkTripSeverity := 500, Cfg_DriveFaultSeverity := 1000, Cfg_IOFaultSeverity := 1000, Cfg_MaxSpdRef := 60.0, Cfg_SpeedRefRawMax := 32767.0, Cfg_SpeedRefEUMax := 130.0, Cfg_SpeedFdbkRawMax := 32767.0, Cfg_SpeedFdbkEUMax := 130.0, Cfg_InpDatalinkRawMax := 4095.0, Cfg_InpDatalinkEUMax := 409.5, Cfg_OutDatalinkMax := 100.0, Cfg_OutDatalinkRawMax := 4095.0, Cfg_OutDatalinkEUMax := 409.5, Cfg_SimRampT := 10, Cfg_FailToStartT := 15, Cfg_FailToStopT := 15, Cfg_ResetPulseT := 2, Val_SpeedRefEUMax := 130.0, Val_SpeedFdbkEUMax := 130.0, Ack_FailToStart := 1, Ack_FailToStop := 1, Ack_IntlkTrip := 1, Ack_DriveFault := 1, Ack_IOFault := 1);
   P_100_B_Intlk_OK : BOOL;
   P_200 : P_VSD := (Inp_Ready := 1, Inp_CommandDir := 1, Inp_ActualDir := 1, Inp_FwdPermOK := 1, Inp_FwdNBPermOK := 1, Inp_RevPermOK := 1, Inp_RevNBPermOK := 1, Inp_IntlkOK := 1, Inp_NBIntlkOK := 1, Cfg_SetTrack := 1, Cfg_PCmdClear := 1, Cfg_ProgDefault := 1, Cfg_ShedOnFailToStart := 1, Cfg_ShedOnIOFault := 1, Cfg_FailToStartAckReqd := 1, Cfg_FailToStopAckReqd := 1, Cfg_IntlkTripAckReqd := 1, Cfg_DriveFaultAckReqd := 1, Cfg_IOFaultAckReqd := 1, Cfg_FailToStartSeverity := 1000, Cfg_FailToStopSeverity := 1000, Cfg_IntlkTripSeverity := 500, Cfg_DriveFaultSeverity := 1000, Cfg_IOFaultSeverity := 1000, Cfg_MaxSpdRef := 60.0, Cfg_SpeedRefRawMax := 32767.0, Cfg_SpeedRefEUMax := 130.0, Cfg_SpeedFdbkRawMax := 32767.0, Cfg_SpeedFdbkEUMax := 130.0, Cfg_InpDatalinkRawMax := 4095.0, Cfg_InpDatalinkEUMax := 409.5, Cfg_OutDatalinkMax := 100.0, Cfg_OutDatalinkRawMax := 4095.0, Cfg_OutDatalinkEUMax := 409.5, Cfg_SimRampT := 10, Cfg_FailToStartT := 15, Cfg_FailToStopT := 15, Cfg_ResetPulseT := 2, Val_SpeedRefEUMax := 130.0, Val_SpeedFdbkEUMax := 130.0, Ack_FailToStart := 1, Ack_FailToStop := 1, Ack_IntlkTrip := 1, Ack_DriveFault := 1, Ack_IOFault := 1);
   P_201 : P_VSD := (Inp_Ready := 1, Inp_CommandDir := 1, Inp_ActualDir := 1, Inp_FwdPermOK := 1, Inp_FwdNBPermOK := 1, Inp_RevPermOK := 1, Inp_RevNBPermOK := 1, Inp_IntlkOK := 1, Inp_NBIntlkOK := 1, Cfg_SetTrack := 1, Cfg_PCmdClear := 1, Cfg_ShedOnFailToStart := 1, Cfg_ShedOnIOFault := 1, Cfg_FailToStartAckReqd := 1, Cfg_FailToStopAckReqd := 1, Cfg_IntlkTripAckReqd := 1, Cfg_DriveFaultAckReqd := 1, Cfg_IOFaultAckReqd := 1, Cfg_FailToStartSeverity := 1000, Cfg_FailToStopSeverity := 1000, Cfg_IntlkTripSeverity := 500, Cfg_DriveFaultSeverity := 1000, Cfg_IOFaultSeverity := 1000, Cfg_MaxSpdRef := 60.0, Cfg_SpeedRefRawMax := 32767.0, Cfg_SpeedRefEUMax := 130.0, Cfg_SpeedFdbkRawMax := 32767.0, Cfg_SpeedFdbkEUMax := 130.0, Cfg_InpDatalinkRawMax := 4095.0, Cfg_InpDatalinkEUMax := 409.5, Cfg_OutDatalinkMax := 100.0, Cfg_OutDatalinkRawMax := 4095.0, Cfg_OutDatalinkEUMax := 409.5, Cfg_SimRampT := 10, Cfg_FailToStartT := 15, Cfg_FailToStopT := 15, Cfg_ResetPulseT := 2, Val_SpeedRefEUMax := 130.0, Val_SpeedFdbkEUMax := 130.0, Ack_FailToStart := 1, Ack_FailToStop := 1, Ack_IntlkTrip := 1, Ack_DriveFault := 1, Ack_IOFault := 1);
   P_202 : P_VSD := (Inp_Ready := 1, Inp_CommandDir := 1, Inp_ActualDir := 1, Inp_FwdPermOK := 1, Inp_FwdNBPermOK := 1, Inp_RevPermOK := 1, Inp_RevNBPermOK := 1, Inp_IntlkOK := 1, Inp_NBIntlkOK := 1, Cfg_SetTrack := 1, Cfg_PCmdClear := 1, Cfg_ShedOnFailToStart := 1, Cfg_ShedOnIOFault := 1, Cfg_FailToStartAckReqd := 1, Cfg_FailToStopAckReqd := 1, Cfg_IntlkTripAckReqd := 1, Cfg_DriveFaultAckReqd := 1, Cfg_IOFaultAckReqd := 1, Cfg_FailToStartSeverity := 1000, Cfg_FailToStopSeverity := 1000, Cfg_IntlkTripSeverity := 500, Cfg_DriveFaultSeverity := 1000, Cfg_IOFaultSeverity := 1000, Cfg_MaxSpdRef := 60.0, Cfg_SpeedRefRawMax := 32767.0, Cfg_SpeedRefEUMax := 130.0, Cfg_SpeedFdbkRawMax := 32767.0, Cfg_SpeedFdbkEUMax := 130.0, Cfg_InpDatalinkRawMax := 4095.0, Cfg_InpDatalinkEUMax := 409.5, Cfg_OutDatalinkMax := 100.0, Cfg_OutDatalinkRawMax := 4095.0, Cfg_OutDatalinkEUMax := 409.5, Cfg_SimRampT := 10, Cfg_FailToStartT := 15, Cfg_FailToStopT := 15, Cfg_ResetPulseT := 2, Val_SpeedRefEUMax := 130.0, Val_SpeedFdbkEUMax := 130.0, Ack_FailToStart := 1, Ack_FailToStop := 1, Ack_IntlkTrip := 1, Ack_DriveFault := 1, Ack_IOFault := 1);
   P_300 : P_VSD := (Inp_Ready := 1, Inp_CommandDir := 1, Inp_ActualDir := 1, Inp_FwdPermOK := 1, Inp_FwdNBPermOK := 1, Inp_RevPermOK := 1, Inp_RevNBPermOK := 1, Inp_IntlkOK := 1, Inp_NBIntlkOK := 1, Cfg_SetTrack := 1, Cfg_PCmdClear := 1, Cfg_ProgDefault := 1, Cfg_ShedOnFailToStart := 1, Cfg_ShedOnIOFault := 1, Cfg_FailToStartAckReqd := 1, Cfg_FailToStopAckReqd := 1, Cfg_IntlkTripAckReqd := 1, Cfg_DriveFaultAckReqd := 1, Cfg_IOFaultAckReqd := 1, Cfg_FailToStartSeverity := 1000, Cfg_FailToStopSeverity := 1000, Cfg_IntlkTripSeverity := 500, Cfg_DriveFaultSeverity := 1000, Cfg_IOFaultSeverity := 1000, Cfg_MaxSpdRef := 60.0, Cfg_SpeedRefRawMax := 32767.0, Cfg_SpeedRefEUMax := 130.0, Cfg_SpeedFdbkRawMax := 32767.0, Cfg_SpeedFdbkEUMax := 130.0, Cfg_InpDatalinkRawMax := 4095.0, Cfg_InpDatalinkEUMax := 409.5, Cfg_OutDatalinkMax := 100.0, Cfg_OutDatalinkRawMax := 4095.0, Cfg_OutDatalinkEUMax := 409.5, Cfg_SimRampT := 10, Cfg_FailToStartT := 15, Cfg_FailToStopT := 15, Cfg_ResetPulseT := 2, Val_SpeedRefEUMax := 130.0, Val_SpeedFdbkEUMax := 130.0, Ack_FailToStart := 1, Ack_FailToStop := 1, Ack_IntlkTrip := 1, Ack_DriveFault := 1, Ack_IOFault := 1);
   P_51A_B : P_Motor := (Inp_PermOK := 1, Inp_NBPermOK := 1, Inp_IntlkOK := 1, Inp_NBIntlkOK := 1, Cfg_PCmdClear := 1, Cfg_ProgDefault := 1, Cfg_ShedOnFailToStart := 1, Cfg_ShedOnIOFault := 1, Cfg_FailToStartAckReqd := 1, Cfg_FailToStopAckReqd := 1, Cfg_IntlkTripAckReqd := 1, Cfg_IOFaultAckReqd := 1, Cfg_FailToStartSeverity := 1000, Cfg_FailToStopSeverity := 1000, Cfg_IntlkTripSeverity := 500, Cfg_IOFaultSeverity := 1000, Cfg_SimFdbkT := 2, Cfg_FailToStartT := 10, Cfg_FailToStopT := 10, Sts_Stopped := 1, Sts_Oper := 1, Ack_FailToStart := 1, Ack_FailToStop := 1, Ack_IntlkTrip := 1, Ack_IOFault := 1);
   P_51A_B_Intlk : P_Intlk := (Cfg_PCmdClear := 1, Sts_IntlkOK := 1, Sts_NBIntlkOK := 1);
   P_51A_BIntlk : P_Intlk := (Cfg_PCmdClear := 1, Sts_IntlkOK := 1, Sts_NBIntlkOK := 1);
   P_Intlk_M_001 : P_Intlk := (Cfg_PCmdClear := 1, Sts_IntlkOK := 1, Sts_NBIntlkOK := 1);
   P_Perm_M_001 : P_Perm := (Inp_Perm00 := 1, Inp_Perm01 := 1, Inp_Perm02 := 1, Inp_Perm03 := 1, Inp_Perm04 := 1, Inp_Perm05 := 1, Inp_Perm06 := 1, Inp_Perm07 := 1, Inp_Perm08 := 1, Inp_Perm09 := 1, Inp_Perm10 := 1, Inp_Perm11 := 1, Inp_Perm12 := 1, Inp_Perm13 := 1, Inp_Perm14 := 1, Inp_Perm15 := 1, Cfg_OKState := 2#1111_1111_1111_1111, Sts_PermOK := 1, Sts_NBPermOK := 1, Sts_Perm := 2#1111_1111_1111_1111);
   PERM_OK_P_51_A_B : BOOL;
   PERM_OK_XV_52 : BOOL;
   PID_Auto_mode : BOOL := 1;
   PID_OUT_TK_200 : REAL := 59.999977;   // Esfuerzo de control Deberá ir direccionada a la salida analogica fisica
   PID_OUT_TK_300 : REAL;
   PID_OUT_TR_100 : REAL;
   PID_TT : PIDE_AUTOTUNE := (ResponseSpeed := 2, PVTuneLimit := 75.0, StepSize := 10.0, TunedGood := 1, ATuneAcquired := 1, UsedProcessType := 7, Gain := 1.0985756, TimeConstant := 5.4, DeadTime := 2.0, PGainTunedFast := 1.8545046, IGainTunedFast := 18.341255, DGainTunedFast := 0.020605609, PGainTunedMed := 1.2363364, IGainTunedMed := 12.227503, DGainTunedMed := 0.013737071, PGainTunedSlow := 0.6181682, IGainTunedSlow := 6.1137514, DGainTunedSlow := 0.0068685357, StepSizeUsed := 10.0);
   PID_TT2 : PIDE_AUTOTUNE;
   PID_TT3 : PIDE_AUTOTUNE;
   PPX_M_100 : P_DescList[1];
   PPX_M_200 : P_DescList[1];
   PPX_M_300 : P_DescList[1];
   PPX_Mixer_VSD_200 : P_DescList[1];
   PPX_P_100_B : P_DescList[1];
   PPX_P_200 : P_DescList[1];
   PPX_P_300 : P_DescList[1];
   PPX_Pump_100_A : P_DescList[1];
   Pump_100_A : P_VSD := (Inp_Ready := 1, Inp_CommandDir := 1, Inp_ActualDir := 1, Inp_FwdPermOK := 1, Inp_FwdNBPermOK := 1, Inp_RevPermOK := 1, Inp_RevNBPermOK := 1, Inp_IntlkOK := 1, Inp_NBIntlkOK := 1, Cfg_SetTrack := 1, Cfg_PCmdClear := 1, Cfg_ProgDefault := 1, Cfg_ShedOnFailToStart := 1, Cfg_ShedOnIOFault := 1, Cfg_FailToStartAckReqd := 1, Cfg_FailToStopAckReqd := 1, Cfg_IntlkTripAckReqd := 1, Cfg_DriveFaultAckReqd := 1, Cfg_IOFaultAckReqd := 1, Cfg_FailToStartSeverity := 1000, Cfg_FailToStopSeverity := 1000, Cfg_IntlkTripSeverity := 500, Cfg_DriveFaultSeverity := 1000, Cfg_IOFaultSeverity := 1000, Cfg_MaxSpdRef := 60.0, Cfg_SpeedRefRawMax := 32767.0, Cfg_SpeedRefEUMax := 130.0, Cfg_SpeedFdbkRawMax := 32767.0, Cfg_SpeedFdbkEUMax := 130.0, Cfg_InpDatalinkRawMax := 4095.0, Cfg_InpDatalinkEUMax := 409.5, Cfg_OutDatalinkMax := 100.0, Cfg_OutDatalinkRawMax := 4095.0, Cfg_OutDatalinkEUMax := 409.5, Cfg_SimRampT := 10, Cfg_FailToStartT := 15, Cfg_FailToStopT := 15, Cfg_ResetPulseT := 2, Val_SpeedRefEUMax := 130.0, Val_SpeedFdbkEUMax := 130.0, Ack_FailToStart := 1, Ack_FailToStop := 1, Ack_IntlkTrip := 1, Ack_DriveFault := 1, Ack_IOFault := 1);
   Pump_100_A1 : P_VSD := (Inp_Ready := 1, Inp_CommandDir := 1, Inp_ActualDir := 1, Inp_FwdPermOK := 1, Inp_FwdNBPermOK := 1, Inp_RevPermOK := 1, Inp_RevNBPermOK := 1, Inp_IntlkOK := 1, Inp_NBIntlkOK := 1, Cfg_SetTrack := 1, Cfg_PCmdClear := 1, Cfg_ShedOnFailToStart := 1, Cfg_ShedOnIOFault := 1, Cfg_FailToStartAckReqd := 1, Cfg_FailToStopAckReqd := 1, Cfg_IntlkTripAckReqd := 1, Cfg_DriveFaultAckReqd := 1, Cfg_IOFaultAckReqd := 1, Cfg_FailToStartSeverity := 1000, Cfg_FailToStopSeverity := 1000, Cfg_IntlkTripSeverity := 500, Cfg_DriveFaultSeverity := 1000, Cfg_IOFaultSeverity := 1000, Cfg_MaxSpdRef := 60.0, Cfg_SpeedRefRawMax := 32767.0, Cfg_SpeedRefEUMax := 130.0, Cfg_SpeedFdbkRawMax := 32767.0, Cfg_SpeedFdbkEUMax := 130.0, Cfg_InpDatalinkRawMax := 4095.0, Cfg_InpDatalinkEUMax := 409.5, Cfg_OutDatalinkMax := 100.0, Cfg_OutDatalinkRawMax := 4095.0, Cfg_OutDatalinkEUMax := 409.5, Cfg_SimRampT := 10, Cfg_FailToStartT := 15, Cfg_FailToStopT := 15, Cfg_ResetPulseT := 2, Val_SpeedRefEUMax := 130.0, Val_SpeedFdbkEUMax := 130.0, Ack_FailToStart := 1, Ack_FailToStop := 1, Ack_IntlkTrip := 1, Ack_DriveFault := 1, Ack_IOFault := 1);
   Pump_100_A_Intlk_Ok : BOOL;
   Pump_100_A_Perm_Ok : BOOL;
   PZT_52 : P_AIn := (Inp_HiHiGate := 1, Inp_HiGate := 1, Inp_LoGate := 1, Inp_LoLoGate := 1, Inp_FailGate := 1, Cfg_SetTrack := 1, Cfg_PCmdClear := 1, Cfg_ProgDefault := 1, Cfg_HiHiAckReqd := 1, Cfg_HiAckReqd := 1, Cfg_LoAckReqd := 1, Cfg_LoLoAckReqd := 1, Cfg_FailAckReqd := 1, Cfg_HiHiSeverity := 750, Cfg_HiSeverity := 500, Cfg_LoSeverity := 500, Cfg_LoLoSeverity := 750, Cfg_FailSeverity := 1000, Cfg_InpRawMin := 3277.0, Cfg_InpRawMax := 16384.0, Cfg_PVEUMax := 100.0, Cfg_HiHiDB := 1.0, Cfg_HiDB := 1.0, Cfg_LoDB := 1.0, Cfg_LoLoDB := 1.0, Cfg_FailHiLim := 103.958336, Cfg_FailLoLim := -2.0833333, Cfg_FailDB := 0.41666666, PSet_HiHiLim := 1.5e+38, PSet_HiLim := 1.5e+38, PSet_LoLim := 5.0, PSet_LoLoLim := -1.5e+38, OSet_HiHiLim := 1.5e+38, OSet_HiLim := 1.5e+38, OSet_LoLim := -1.5e+38, OSet_LoLoLim := -1.5e+38, Val_PVMinCapt := 1.5e+38, Val_PVMaxCapt := -1.5e+38, Val_PVEUMax := 100.0, Val_HiHiLim := 1.5e+38, Val_HiLim := 1.5e+38, Val_LoLim := -1.5e+38, Val_LoLoLim := -1.5e+38, Sts_InpPV := 1, Sts_Oper := 1, Ack_HiHi := 1, Ack_Hi := 1, Ack_Lo := 1, Ack_LoLo := 1, Ack_Fail := 1);
   PZT_53 : P_AIn := (Inp_HiHiGate := 1, Inp_HiGate := 1, Inp_LoGate := 1, Inp_LoLoGate := 1, Inp_FailGate := 1, Cfg_SetTrack := 1, Cfg_PCmdClear := 1, Cfg_HiHiAckReqd := 1, Cfg_HiAckReqd := 1, Cfg_LoAckReqd := 1, Cfg_LoLoAckReqd := 1, Cfg_FailAckReqd := 1, Cfg_HiHiSeverity := 750, Cfg_HiSeverity := 500, Cfg_LoSeverity := 500, Cfg_LoLoSeverity := 750, Cfg_FailSeverity := 1000, Cfg_InpRawMin := 3277.0, Cfg_InpRawMax := 16384.0, Cfg_PVEUMax := 100.0, Cfg_HiHiDB := 1.0, Cfg_HiDB := 1.0, Cfg_LoDB := 1.0, Cfg_LoLoDB := 1.0, Cfg_FailHiLim := 103.958336, Cfg_FailLoLim := -2.0833333, Cfg_FailDB := 0.41666666, PSet_HiHiLim := 1.5e+38, PSet_HiLim := 1.5e+38, PSet_LoLim := 95.0, PSet_LoLoLim := -1.5e+38, OSet_HiHiLim := 1.5e+38, OSet_HiLim := 1.5e+38, OSet_LoLim := -1.5e+38, OSet_LoLoLim := -1.5e+38, Val_PVMinCapt := 1.5e+38, Val_PVMaxCapt := -1.5e+38, Val_PVEUMax := 100.0, Val_HiHiLim := 1.5e+38, Val_HiLim := 1.5e+38, Val_LoLim := -1.5e+38, Val_LoLoLim := -1.5e+38, Sts_InpPV := 1, Sts_Oper := 1, Ack_HiHi := 1, Ack_Hi := 1, Ack_Lo := 1, Ack_LoLo := 1, Ack_Fail := 1);
   realimentacion : BOOL;
   SET_POINT_2_Temperatura : REAL;
   SET_POINT_3_Temperatura : REAL;
   SET_POINT_Temperatura : REAL;
   SP_Timer_M_100 : TIMER := (PRE := 20000);
   SP_Timer_Mix : TIMER := (PRE := 30000);
   Sp_Timer_P_200 : TIMER := (PRE := 30000);
   SP_Timer_P_300 : TIMER := (PRE := 40000);
   SP_veloc_M2 : DINT := 20;
   Sp_veloc_M_200 : DINT := 68;
   SP_veloc_Mix : DINT := 20;
   SP_veloc_P_100_B : DINT := 70;
   SP_veloc_Pump_100_A : DINT := 60;
   TCV_100 : P_ValveC := (Inp_IntlkOK := 1, Inp_NBIntlkOK := 1, Cfg_ShedOnIOFault := 1, Cfg_SetTrack := 1, Cfg_LSFail := 1, Cfg_PCmdClear := 1, Cfg_IntlkTripAckReqd := 1, Cfg_ActuatorFaultAckReqd := 1, Cfg_IOFaultAckReqd := 1, Cfg_IntlkTripSeverity := 500, Cfg_ActuatorFaultSeverity := 1000, Cfg_IOFaultSeverity := 1000, Cfg_MaxCV := 100.0, Cfg_MaxCVRoCInc := 10.0, Cfg_MaxCVRoCDec := 10.0, Cfg_CVEUMax := 100.0, Cfg_CVRawMin := 3277.0, Cfg_CVRawMax := 16384.0, Cfg_FdbkRawMax := 100.0, Cfg_CycleT := 10.0, Cfg_OpenRate := 1.0, Cfg_CloseRate := 1.0, Cfg_MaxOnT := 5.0, Cfg_MinOnT := 1.0, Val_CVEUMax := 100.0, Ack_IntlkTrip := 1, Ack_ActuatorFault := 1, Ack_IOFault := 1);
   TCV_101 : P_ValveC := (Inp_IntlkOK := 1, Inp_NBIntlkOK := 1, Cfg_ShedOnIOFault := 1, Cfg_SetTrack := 1, Cfg_LSFail := 1, Cfg_PCmdClear := 1, Cfg_IntlkTripAckReqd := 1, Cfg_ActuatorFaultAckReqd := 1, Cfg_IOFaultAckReqd := 1, Cfg_IntlkTripSeverity := 500, Cfg_ActuatorFaultSeverity := 1000, Cfg_IOFaultSeverity := 1000, Cfg_MaxCV := 100.0, Cfg_MaxCVRoCInc := 10.0, Cfg_MaxCVRoCDec := 10.0, Cfg_CVEUMax := 100.0, Cfg_CVRawMin := 3277.0, Cfg_CVRawMax := 16384.0, Cfg_FdbkRawMax := 100.0, Cfg_CycleT := 10.0, Cfg_OpenRate := 1.0, Cfg_CloseRate := 1.0, Cfg_MaxOnT := 5.0, Cfg_MinOnT := 1.0, Val_CVEUMax := 100.0, Ack_IntlkTrip := 1, Ack_ActuatorFault := 1, Ack_IOFault := 1);
   TCV_200 : P_ValveC := (Inp_IntlkOK := 1, Inp_NBIntlkOK := 1, Cfg_ShedOnIOFault := 1, Cfg_SetTrack := 1, Cfg_LSFail := 1, Cfg_PCmdClear := 1, Cfg_ProgDefault := 1, Cfg_IntlkTripAckReqd := 1, Cfg_ActuatorFaultAckReqd := 1, Cfg_IOFaultAckReqd := 1, Cfg_IntlkTripSeverity := 500, Cfg_ActuatorFaultSeverity := 1000, Cfg_IOFaultSeverity := 1000, Cfg_MaxCV := 100.0, Cfg_MaxCVRoCInc := 10.0, Cfg_MaxCVRoCDec := 10.0, Cfg_CVEUMax := 100.0, Cfg_CVRawMax := 100.0, Cfg_FdbkRawMax := 100.0, Cfg_CycleT := 10.0, Cfg_OpenRate := 1.0, Cfg_CloseRate := 1.0, Cfg_MaxOnT := 5.0, Cfg_MinOnT := 1.0, Val_CVEUMax := 100.0, Ack_IntlkTrip := 1, Ack_ActuatorFault := 1, Ack_IOFault := 1);
   TCV_300 : P_ValveC := (Inp_IntlkOK := 1, Inp_NBIntlkOK := 1, Cfg_ShedOnIOFault := 1, Cfg_SetTrack := 1, Cfg_LSFail := 1, Cfg_PCmdClear := 1, Cfg_ProgDefault := 1, Cfg_IntlkTripAckReqd := 1, Cfg_ActuatorFaultAckReqd := 1, Cfg_IOFaultAckReqd := 1, Cfg_IntlkTripSeverity := 500, Cfg_ActuatorFaultSeverity := 1000, Cfg_IOFaultSeverity := 1000, Cfg_MaxCV := 100.0, Cfg_MaxCVRoCInc := 10.0, Cfg_MaxCVRoCDec := 10.0, Cfg_CVEUMax := 100.0, Cfg_CVRawMax := 100.0, Cfg_FdbkRawMax := 100.0, Cfg_CycleT := 10.0, Cfg_OpenRate := 1.0, Cfg_CloseRate := 1.0, Cfg_MaxOnT := 5.0, Cfg_MinOnT := 1.0, Val_CVEUMax := 100.0, Ack_IntlkTrip := 1, Ack_ActuatorFault := 1, Ack_IOFault := 1);
   Temperatura_ok : BOOL;
   Temperatura_TR_100 : REAL;
   Temperatura_TT_100 : REAL := 59.99998;   // Variable del proceso Deberá ir direccionada a la entrada analogica fisica
   Temperatura_TT_200 : REAL;
   Temperatura_TT_300 : REAL;
   Timer_molienda_ctrlTemp : TIMER := (PRE := 60000);
   TK_100_Lleno : BOOL;
   TT_100 : P_AIn := (Inp_HiHiGate := 1, Inp_HiGate := 1, Inp_LoGate := 1, Inp_LoLoGate := 1, Inp_FailGate := 1, Cfg_SetTrack := 1, Cfg_PCmdClear := 1, Cfg_HiHiAckReqd := 1, Cfg_HiAckReqd := 1, Cfg_LoAckReqd := 1, Cfg_LoLoAckReqd := 1, Cfg_FailAckReqd := 1, Cfg_HiHiSeverity := 750, Cfg_HiSeverity := 500, Cfg_LoSeverity := 500, Cfg_LoLoSeverity := 750, Cfg_FailSeverity := 1000, Cfg_InpRawMax := 100.0, Cfg_PVEUMax := 100.0, Cfg_HiHiDB := 1.0, Cfg_HiDB := 1.0, Cfg_LoDB := 1.0, Cfg_LoLoDB := 1.0, Cfg_FailHiLim := 103.958336, Cfg_FailLoLim := -2.0833333, Cfg_FailDB := 0.41666666, PSet_HiHiLim := 1.5e+38, PSet_HiLim := 1.5e+38, PSet_LoLim := -1.5e+38, PSet_LoLoLim := -1.5e+38, OSet_HiHiLim := 1.5e+38, OSet_HiLim := 1.5e+38, OSet_LoLim := -1.5e+38, OSet_LoLoLim := -1.5e+38, Val_PVMinCapt := 1.5e+38, Val_PVMaxCapt := -1.5e+38, Val_PVEUMax := 100.0, Val_HiHiLim := 1.5e+38, Val_HiLim := 1.5e+38, Val_LoLim := -1.5e+38, Val_LoLoLim := -1.5e+38, Sts_InpPV := 1, Sts_Oper := 1, Ack_HiHi := 1, Ack_Hi := 1, Ack_Lo := 1, Ack_LoLo := 1, Ack_Fail := 1);
   TT_101 : P_AIn := (Inp_HiHiGate := 1, Inp_HiGate := 1, Inp_LoGate := 1, Inp_LoLoGate := 1, Inp_FailGate := 1, Cfg_SetTrack := 1, Cfg_PCmdClear := 1, Cfg_HiHiAckReqd := 1, Cfg_HiAckReqd := 1, Cfg_LoAckReqd := 1, Cfg_LoLoAckReqd := 1, Cfg_FailAckReqd := 1, Cfg_HiHiSeverity := 750, Cfg_HiSeverity := 500, Cfg_LoSeverity := 500, Cfg_LoLoSeverity := 750, Cfg_FailSeverity := 1000, Cfg_InpRawMax := 100.0, Cfg_PVEUMax := 100.0, Cfg_HiHiDB := 1.0, Cfg_HiDB := 1.0, Cfg_LoDB := 1.0, Cfg_LoLoDB := 1.0, Cfg_FailHiLim := 103.958336, Cfg_FailLoLim := -2.0833333, Cfg_FailDB := 0.41666666, PSet_HiHiLim := 1.5e+38, PSet_HiLim := 1.5e+38, PSet_LoLim := -1.5e+38, PSet_LoLoLim := -1.5e+38, OSet_HiHiLim := 1.5e+38, OSet_HiLim := 1.5e+38, OSet_LoLim := -1.5e+38, OSet_LoLoLim := -1.5e+38, Val_PVMinCapt := 1.5e+38, Val_PVMaxCapt := -1.5e+38, Val_PVEUMax := 100.0, Val_HiHiLim := 1.5e+38, Val_HiLim := 1.5e+38, Val_LoLim := -1.5e+38, Val_LoLoLim := -1.5e+38, Sts_InpPV := 1, Sts_Oper := 1, Ack_HiHi := 1, Ack_Hi := 1, Ack_Lo := 1, Ack_LoLo := 1, Ack_Fail := 1);
   TT_102 : P_AIn := (Inp_HiHiGate := 1, Inp_HiGate := 1, Inp_LoGate := 1, Inp_LoLoGate := 1, Inp_FailGate := 1, Cfg_SetTrack := 1, Cfg_PCmdClear := 1, Cfg_HiHiAckReqd := 1, Cfg_HiAckReqd := 1, Cfg_LoAckReqd := 1, Cfg_LoLoAckReqd := 1, Cfg_FailAckReqd := 1, Cfg_HiHiSeverity := 750, Cfg_HiSeverity := 500, Cfg_LoSeverity := 500, Cfg_LoLoSeverity := 750, Cfg_FailSeverity := 1000, Cfg_InpRawMax := 100.0, Cfg_PVEUMax := 100.0, Cfg_HiHiDB := 1.0, Cfg_HiDB := 1.0, Cfg_LoDB := 1.0, Cfg_LoLoDB := 1.0, Cfg_FailHiLim := 103.958336, Cfg_FailLoLim := -2.0833333, Cfg_FailDB := 0.41666666, PSet_HiHiLim := 1.5e+38, PSet_HiLim := 1.5e+38, PSet_LoLim := -1.5e+38, PSet_LoLoLim := -1.5e+38, OSet_HiHiLim := 1.5e+38, OSet_HiLim := 1.5e+38, OSet_LoLim := -1.5e+38, OSet_LoLoLim := -1.5e+38, Val_PVMinCapt := 1.5e+38, Val_PVMaxCapt := -1.5e+38, Val_PVEUMax := 100.0, Val_HiHiLim := 1.5e+38, Val_HiLim := 1.5e+38, Val_LoLim := -1.5e+38, Val_LoLoLim := -1.5e+38, Sts_InpPV := 1, Sts_Oper := 1, Ack_HiHi := 1, Ack_Hi := 1, Ack_Lo := 1, Ack_LoLo := 1, Ack_Fail := 1);
   XV_52 : P_ValveSO := (Inp_PermOK := 1, Inp_NBPermOK := 1, Inp_IntlkOK := 1, Inp_NBIntlkOK := 1, Cfg_LSFail := 1, Cfg_PCmdClear := 1, Cfg_ProgDefault := 1, Cfg_ShedOnFullStall := 1, Cfg_ShedOnTransitStall := 1, Cfg_ShedOnIOFault := 1, Cfg_FullStallAckReqd := 1, Cfg_TransitStallAckReqd := 1, Cfg_IntlkTripAckReqd := 1, Cfg_IOFaultAckReqd := 1, Cfg_FullStallSeverity := 1000, Cfg_TransitStallSeverity := 1000, Cfg_IntlkTripSeverity := 500, Cfg_IOFaultSeverity := 1000, Cfg_SimFdbkT := 2, Cfg_FullStallT := 5, Cfg_TransitStallT := 10, Ack_FullStall := 1, Ack_TransitStall := 1, Ack_IntlkTrip := 1, Ack_IOFault := 1);
END_VAR
